IF reversePolarity THEN
    distanceToMoveInSteps := distanceToMoveInSteps * -1;
END_IF

pointToPointAccelSetpoint := acceleration;
pointToPointDecelSetpoint := deceleration;
velocitySetpoint := velocity;

currentLimit := defaultCurrentSetpoint;
_moveDistance := TRUE;

//commands.feedToLength := TRUE;
//SUPER^.ExecuteStoredProgram(1);
END_METHOD

METHOD StopViaProgram
// Load program segment 12 into buffer and execute.  This program contains nothing but a SM command.
// We must do it this way because the normal "stop command" opcode we have access to over modbus 
// also kills the program buffer which is bad.
SUPER^.Stop();
END_METHOD

PROPERTY CommandAcknowledged : BOOL
GET
CommandAcknowledged := _moveDone;
END_GET
END_PROPERTY

METHOD SetTorque
VAR_INPUT
	torque : DINT;
END_VAR
sclCommand := 16#4743; // GC (Current Command)
parameter1 := torque;
															
commandSuccessful := FALSE;
commands.SendHostCommand := TRUE;
END_METHOD

METHOD Execute
VAR_INPUT
END_VAR
SUPER^.Execute();
waitForMove();
_moveDistanceONS(CLK := _moveDistance);
_moveFinalONS(CLK := _moveFinal);

CASE moveDistanceState OF
	AMP_EIP_MOVE_INITIAL_STATES.Idle :						
															IF _moveDistance THEN
																moveDistanceState := AMP_EIP_MOVE_INITIAL_STATES.SetOutputOff;
															END_IF
															
	AMP_EIP_MOVE_INITIAL_STATES.SetOutputOff :					sclCommand := 16#534F; //Output off
															parameter1 := 16#48B2;
															commands.SendHostCommand := TRUE;
															IF commandSuccessful THEN
																commandSuccessful := FALSE;
																moveDistanceState := AMP_EIP_MOVE_INITIAL_STATES.WaitAfterSettingOutputOff;
															END_IF
															
	AMP_EIP_MOVE_INITIAL_STATES.WaitAfterSettingOutputOff :		
															IF commandSuccessful THEN
																moveDistanceState := AMP_EIP_MOVE_INITIAL_STATES.MoveMotor;
															END_IF
																
	AMP_EIP_MOVE_INITIAL_STATES.MoveMotor: 					commandSuccessful := FALSE;
															sclCommand := 16#0;
															parameter1 := 16#0;
															commands.FeedToLength := TRUE;
															_moveDistance := FALSE;
															moveDistanceState := AMP_EIP_MOVE_INITIAL_STATES.WaitAfterMovingMotor;
															
															
	AMP_EIP_MOVE_INITIAL_STATES.WaitAfterMovingMotor: 		IF commandSuccessful THEN
																_moveDone := TRUE;
																moveDistanceState := AMP_EIP_MOVE_INITIAL_STATES.Idle;
															END_IF														
END_CASE

CASE moveDistanceFinalState OF
	AMP_EIP_MOVE_INITIAL_STATES.Idle :						IF _moveFinal THEN
																moveDistanceFinalState := AMP_EIP_MOVE_INITIAL_STATES.SetOutputOff;
															END_IF
															
	AMP_EIP_MOVE_INITIAL_STATES.SetOutputOff :					sclCommand := 16#534F; //Output off
															parameter1 := 16#48B2;
															commands.SendHostCommand := TRUE;
															IF commandSuccessful THEN
																commandSuccessful := FALSE;
																moveDistanceFinalState := AMP_EIP_MOVE_INITIAL_STATES.WaitAfterSettingOutputOff;
															END_IF
															
	AMP_EIP_MOVE_INITIAL_STATES.WaitAfterSettingOutputOff :		
															IF commandSuccessful THEN
																moveDistanceFinalState := AMP_EIP_MOVE_INITIAL_STATES.MoveMotor;
															END_IF
															
	AMP_EIP_MOVE_INITIAL_STATES.MoveMotor: 					sclCommand := 16#0;
															parameter1 := 16#0;
															commandSuccessful := FALSE;	
															commands.FeedToLength := TRUE;
															moveDistanceFinalState := AMP_EIP_MOVE_INITIAL_STATES.WaitAfterMovingMotor;
															
															
	AMP_EIP_MOVE_INITIAL_STATES.WaitAfterMovingMotor: 		IF commandSuccessful AND InPosition THEN	
																moveDistanceFinalState := AMP_EIP_MOVE_INITIAL_STATES.SetOutputOn;
															END_IF
														
	AMP_EIP_MOVE_INITIAL_STATES.SetOutputOn :					sclCommand := 16#534F; // Output on
															parameter1 := 16#4CB2;
															
															commandSuccessful := FALSE;
															commands.SendHostCommand := TRUE;
															_moveFinal := FALSE;
															moveDistanceFinalState := AMP_EIP_MOVE_INITIAL_STATES.WaitAfterSettingOutputOn;
															
															
	AMP_EIP_MOVE_INITIAL_STATES.WaitAfterSettingOutputOn :		
															IF commandSuccessful THEN
																_moveDone := TRUE;
																moveDistanceFinalState := AMP_EIP_MOVE_INITIAL_STATES.Idle;
															END_IF
																

END_CASE
(*
IF _moveFinal THEN	
	IF NOT movedFinal AND commandSuccessful THEN
		commandSuccessful := FALSE;
		commands.FeedToLength := TRUE;
		waitForMove.IN := TRUE;
		movedFinal := TRUE;
	END_IF
	
	IF commandSuccessful AND waitForMove.Q AND InPosition THEN
		sclCommand := 16#534F;
		parameter1 := 16#4CB2;
		commands.SendHostCommand := TRUE;
		_moveFinal := FALSE;
		waitForMove.IN := FALSE;
		movedFinal := FALSE;
	END_IF
END_IF
*)
IF manualFinalMovePB THEN
    MoveDistanceFinal(distance := distanceSetpointInches, acceleration := pointToPointAccelSetpoint, deceleration := pointToPointDecelSetpoint, velocity := velocitySetpoint);
    manualFinalMovePB := FALSE;
END_IF
END_METHOD

METHOD SetRearMotorTorqueValue
VAR_INPUT
	torque : DINT;
END_VAR
sclCommand := 16#4743; // GC (Current Command)
parameter1 := torque;
															
commandSuccessful := FALSE;
commands.SendHostCommand := TRUE;
END_METHOD

METHOD MoveDistanceFinal
VAR_INPUT
    distance : REAL;        //Distance to move in inches
    acceleration : INT;        //Acceleration in RPM/sec
    deceleration : INT;        //Deceleration in RPM/sec
    velocity : INT;            //Velocity in .25RPM
END_VAR
commandSuccessful := FALSE;
_moveDone := FALSE;
moveDistanceFinalState := AMP_EIP_MOVE_INITIAL_STATES.Idle;
distanceToMoveInSteps := REAL_TO_DINT((distance) * stepsPerInchSetpoint);
IF reversePolarity THEN
    distanceToMoveInSteps := distanceToMoveInSteps * -1;
END_IF

pointToPointAccelSetpoint := acceleration;
pointToPointDecelSetpoint := deceleration;
velocitySetpoint := velocity;

currentLimit := defaultCurrentSetpoint;
_moveFinal := TRUE;
//SUPER^.ExecuteStoredProgram(2);
END_METHOD

END_FUNCTION_BLOCK

// FBs/Motors/Applied Motion/FB_AppliedMotionStepServoEIPBase
FUNCTION_BLOCK FB_AppliedMotionStepServoEIPBase IMPLEMENTS IPositionableMotor
VAR_INPUT
    ptrEIPInputs : POINTER TO ARRAY[0..13] OF  DINT;
    ptrEIPOutputs : POINTER TO ARRAY[0..15] OF DINT;
	commFail : BOOL;
    stepsPerInchSetpoint : INT;             //Steps per inch setpoint
    reversePolarity : BOOL;                 //0 = Normal, 1 = reversed polarity for display
    jogAccelSetpoint : INT;        //Point-to-Point Acceleration (AC) Setpoint
    jogDecelSetpoint : INT;        //Point-to-Point Deceleration (DE) Setpoint
    jogVelocitySetpoint : INT;                //Velocity (VE) Setpoint
    pointToPointAccelSetpoint : INT;        //Point-to-Point Acceleration (AC) Setpoint
    pointToPointDecelSetpoint : INT;        //Point-to-Point Deceleration (DE) Setpoint
    velocitySetpoint : INT;                //Velocity (VE) Setpoint
	defaultCurrentSetpoint : DINT;
	sclCommand : DINT;						// SCL Command from 
	parameter1 : DINT;						// Data/SCL parameter 1
	parameter2 : DINT;						// Data/SCL parameter 2
    distanceSetpointInches : REAL;        //Distance setpoint in inches Setpoint
    moveDistanceManualPB : BOOL;            //Move distance pushbutton
    movePositionManualPB : BOOL;            //Move position pushbutton
	isHomable : BOOL;
END_VAR
VAR_IN_OUT
    //slave : IoDrvModbusTCP.ModbusTCPSlave;                    //Slave ModbusTCP Object
END_VAR
VAR
    absolutePositionSteps : DINT; //Immediate Absolute Position in steps
    distanceToMoveInSteps : DINT;        //Distance Setpoint to Drive
    stepServoStatusRaw : INT; //Raw step servo status over modbus
	stepServoAlarmCodeRaw : INT; // Ras Step Servo alarm code word
	currentLimit : DINT;
    commands : FB_StepServoCommands();
    commandSuccessful : BOOL;    //Modbus Command was successful
    commandSuccessfulONS : R_TRIG;    //Modbus Command was successful
    commandSentONS : R_TRIG;    //Modbus Command was successful
    homeRequiredIndication : BOOL; //Home required indication.
    driveInputs : ARRAY[0..13] OF DINT;        // Inputs from drive over EIP
    driveOutputs : ARRAY[0..15] OF DINT;    // Outputs to drive over EIP
    interfaceToPass : IFault;
    faultListRegisterSuccess : BOOL;        // Registering in fault list successful
    _faulted : BOOL;                    // Motor Faulted
	_reset : BOOL;			//Reset Motor
	_homeNow : BOOL;
	homingOSF : F_TRIG;
	resetState : INT;
	IECReferenceGood : BOOL;
	resetTimeout : Standard.TON;
	encoderResetTimeout : Standard.TON;
END_VAR
VAR_OUTPUT
    absolutePositonInches : REAL; //Immediate Absolute Positon in inches
    velocity : INT;    //Velocity (VE) Input from Drive
    status : StepServoStatusFB; //Status of servo
	alarms : FB_StepServoAlarms; // Alarms from Drive
    QSegmentRunning : INT; //Current Q program running from Drive
	faults : StepServoFaultsType;
END_VAR

//{warning 'add method implementation '}
METHOD Stop
commandSuccessful := FALSE;
commands.StopNormal := TRUE;
END_METHOD

{attribute 'monitoring' := 'variable'}
PROPERTY Homing : BOOL
GET
Homing := status.homing;
END_GET
END_PROPERTY

METHOD HomeNow
commandSuccessful := FALSE;
parameter1 := 1;
pointToPointAccelSetpoint := 50;
pointToPointDecelSetpoint := 50;
velocitySetpoint := 500;
distanceToMoveInSteps := 0;
commands.sendQAndExecute := TRUE;

//homeRequiredIndication := FALSE;
END_METHOD

METHOD MoveDistance
VAR_INPUT
    (*Distance to move in inches*)
    distance    : REAL;
    (*Acceleration in RPM/sec*)
    acceleration    : INT;
    (*Deceleration in RPM/sec*)
    deceleration    : INT;
    (*Velocity in .25RPM*)
    velocity    : INT;
END_VAR
//This method preps the data to send to the drive and triggers the send.
//Set distance and unpack to prep data to send to motor

commandSuccessful := FALSE;

distanceToMoveInSteps := REAL_TO_DINT((distance) * stepsPerInchSetpoint);
IF reversePolarity THEN
    distanceToMoveInSteps := distanceToMoveInSteps * -1;
END_IF

pointToPointAccelSetpoint := acceleration;
pointToPointDecelSetpoint := deceleration;
velocitySetpoint := velocity;
currentLimit := defaultCurrentSetpoint;

commands.feedToLength := TRUE;
END_METHOD

{attribute 'monitoring' := 'variable'}
PROPERTY CommandAcknowledged : BOOL
GET
CommandAcknowledged := commandSuccessful;
END_GET
END_PROPERTY

PROPERTY InstanceName : STRING
GET
END_GET
SET
END_SET
END_PROPERTY

(* This will be called if the machine is faulted*)
METHOD MachineFaulted
END_METHOD

METHOD MoveToPositionTorque
VAR_INPUT
	(*Position to move to in inches*)
    position    : REAL;
    (*Acceleration in RPM/sec*)
    acceleration    : INT;
    (*Deceleration in RPM/sec*)
    deceleration    : INT;
    (*Velocity in .25RPM*)
    velocity    : INT;
	(*Current in .01A*)
	current : DINT;
END_VAR
commandSuccessful := FALSE;

distanceToMoveInSteps := REAL_TO_DINT((position) * stepsPerInchSetpoint);
IF reversePolarity THEN
    distanceToMoveInSteps := distanceToMoveInSteps * -1;    
END_IF

pointToPointAccelSetpoint := acceleration;
pointToPointDecelSetpoint := deceleration;
velocitySetpoint := velocity;
currentLimit := current;

commands.feedToPosition := TRUE;
END_METHOD

{attribute 'monitoring' := 'variable'}
PROPERTY InPosition : BOOL
GET
InPosition := status.inPosition;
END_GET
END_PROPERTY

//{warning 'add method implementation '}
METHOD Disable
commandSuccessful := FALSE;
commands.Disable := TRUE;
END_METHOD

//{warning 'add method implementation '}
METHOD Enable
commandSuccessful := FALSE;
commands.Enable := TRUE;
END_METHOD

METHOD ResetEncoderPosition
VAR_INPUT
	position : DINT;
END_VAR
sclCommand := 16#5350; // SP (Set Position)
parameter1 := position;
															
commandSuccessful := FALSE;
commands.SendHostCommand := TRUE;
END_METHOD

METHOD Execute
VAR_INPUT
END_VAR
//    Function Block: AppliedMotionStepServo
//    Description: This block provides an abstraction for a Ethernet I/P Applied Motion Step Servo
//    Created by: Ben Hess
//    Created Date: May 11th, 2018

// Use pointers for EIP memory register locations
driveInputs := ptrEIPInputs^;
// Step servo command bits handler
commands();
ptrEIPOutputs^ := driveOutputs;
alarms(alarmCode := stepServoAlarmCodeRaw, faults := faults);

IF currentLimit = 0 THEN 
	currentLimit := defaultCurrentSetpoint;
END_IF
//Map raw EIP Registers to parameters
absolutePositionSteps := driveInputs[5];
velocity := DINT_TO_INT(driveInputs[8]);
stepServoStatusRaw := DINT_TO_INT(driveInputs[0]);
stepServoAlarmCodeRaw := DINT_TO_INT(driveInputs[1]);
driveOutputs[4] := velocitySetpoint;
driveOutputs[5] := pointToPointAccelSetpoint;
driveOutputs[6] := pointToPointDecelSetpoint;
driveOutputs[7] := distanceToMoveInSteps;
driveOutputs[8] := currentLimit;
driveOutputs[9] := sclCommand;
driveOutputs[10] := parameter1;
driveOutputs[11] := parameter2;
driveOutputs[12] := currentLimit;
driveOutputs[13] := currentLimit;
driveOutputs[0] := commands.commandWord;

//Convert Distance setpoint to steps.  Reverse polarity for display purposes if needed. 

absolutePositonInches := (DINT_TO_REAL(absolutePositionSteps) / INT_TO_REAL(stepsPerInchSetpoint));

//Homing required from motor - for now just if there was an initialization seen.
homeRequiredIndication S= status.initializing OR Globals.firstScan OR _faulted OR driveInputs[11].0;
//homeRequiredIndication S= status.initializing OR Globals.firstScan OR driveInputs[11].0;
homingOSF(CLK := status.homing);
IF NOT driveInputs[11].0 THEN
	homeRequiredIndication := FALSE;
END_IF

commandSentONS(CLK := commands.commandSent);

IF commandSentONS.Q THEN
	commandSuccessful := TRUE;
END_IF

commandSuccessfulONS(CLK := commandSuccessful);
IF commandSuccessfulONS.Q THEN
	//parameter1 := 0;
	//velocitySetpoint := 0;
	//pointToPointAccelSetpoint := 0;
	//pointToPointDecelSetpoint := 0;
	//distanceToMoveInSteps := 0;
END_IF



resetTimeout(IN := _reset, PT := T#1S);
encoderResetTimeout(PT := T#150MS);
IF resetTimeout.Q THEN
	resetState := 0;
	encoderResetTimeout.IN := FALSE;
	_reset := FALSE;
END_IF
CASE resetState OF
	
	0 :		// Do Nothing
			IF _reset THEN
				resetState := 1;
			END_IF
	1 :		// 
			commandSuccessful := FALSE;
			commands.alarmReset := TRUE;
			resetState := 2;
	
	2 :		IF commandSuccessful THEN
				commandSuccessful := FALSE;
				commands.Enable := TRUE;
				resetState := 3;		
			END_IF
	
	3 :		//
			IF commandSuccessful THEN;
				
				encoderResetTimeout.IN := TRUE;
				IF encoderResetTimeout.Q THEN
					resetState := 4;	
					ResetEncoderPosition(driveInputs[5]);	
				END_IF
			END_IF
	
	4 :		//
			IF commandSuccessful THEN;
				resetState := 0;
				
				_reset := FALSE;
			END_IF
	
END_CASE

IF reversePolarity THEN
    absolutePositonInches := absolutePositonInches * -1; 
END_IF

//Get Servo Status and unpack
status(statusCode := StepServoStatusRaw);

//Bit-packing for LONG types over Modbus
//_faulted := status.driveFaulted OR status.alarmPresent OR commFail;
_faulted := status.driveFaulted OR commFail;

//Manual moves for motor
IF moveDistanceManualPB THEN
    MoveDistance(distance := distanceSetpointInches, acceleration := pointToPointAccelSetpoint, deceleration := pointToPointDecelSetpoint, velocity := velocitySetpoint);
    moveDistanceManualPB := FALSE;
END_IF

IF movePositionManualPB THEN
    MoveToPosition(position := distanceSetpointInches, acceleration := pointToPointAccelSetpoint, deceleration := pointToPointDecelSetpoint, velocity := velocitySetpoint);
    movePositionManualPB := FALSE;
END_IF


faults.commFail.faultTrigger := commFail; //AND Globals.machinePowerOK;
//faults.notHomed.faultTrigger := homeRequiredIndication AND isHomable;
END_METHOD

{attribute 'monitoring' := 'variable'}
PROPERTY HomeRequired : BOOL
SET
homeRequiredIndication := HomeRequired;
END_SET
GET
HomeRequired := homeRequiredIndication;
END_GET
END_PROPERTY

{attribute 'monitoring' := 'variable'}
PROPERTY ActiveStoredProgramNumber : INT
GET
ActiveStoredProgramNumber := QSegmentRunning;
END_GET
END_PROPERTY

METHOD Reset : BOOL
VAR_INPUT
END_VAR
_reset := TRUE;
END_METHOD

{attribute 'monitoring' := 'variable'}
PROPERTY Faulted : BOOL
GET
Faulted := _faulted;
END_GET
SET
END_SET
END_PROPERTY

METHOD MoveToPosition
VAR_INPUT
    (*Position to move to in inches*)
    position    : REAL;
    (*Acceleration in RPM/sec*)
    acceleration    : INT;
    (*Deceleration in RPM/sec*)
    deceleration    : INT;
    (*Velocity in .25RPM*)
    velocity    : INT;
END_VAR
commandSuccessful := FALSE;

distanceToMoveInSteps := REAL_TO_DINT((position) * stepsPerInchSetpoint);
IF reversePolarity THEN
    distanceToMoveInSteps := distanceToMoveInSteps * -1;    
END_IF

pointToPointAccelSetpoint := acceleration;
pointToPointDecelSetpoint := deceleration;
velocitySetpoint := velocity;
currentLimit := defaultCurrentSetpoint;

commands.feedToPosition := TRUE;
END_METHOD

METHOD SetTorque
VAR_INPUT
	torque : DINT;
END_VAR
sclCommand := 16#4743; // GC (Current Command)
parameter1 := torque;
															
commandSuccessful := FALSE;
commands.SendHostCommand := TRUE;
END_METHOD

METHOD ExecuteStoredProgram
VAR_INPUT
    (*Program number to execute*)
    programNumber    : INT;
END_VAR
parameter1 := programNumber;
commands.SendQAndExecute := TRUE;
END_METHOD

{attribute 'monitoring' := 'variable'}
PROPERTY CurrentPosition : REAL  //Current motor position in Inches
GET
CurrentPosition := absolutePositonInches;
END_GET
END_PROPERTY

{attribute 'monitoring' := 'variable'}
PROPERTY Moving : BOOL
GET
Moving := status.moving;
END_GET
END_PROPERTY

METHOD MoveDistanceTorque
VAR_INPUT
	(*Distance to move in inches*)
    distance    : REAL;
    (*Acceleration in RPM/sec*)
    acceleration    : INT;
    (*Deceleration in RPM/sec*)
    deceleration    : INT;
    (*Velocity in .25RPM*)
    velocity    : INT;
	(*Current in .01A*)
	current : DINT;
END_VAR
//This method preps the data to send to the drive and triggers the send.
//Set distance and unpack to prep data to send to motor

commandSuccessful := FALSE;

distanceToMoveInSteps := REAL_TO_DINT((distance) * stepsPerInchSetpoint);
IF reversePolarity THEN
    distanceToMoveInSteps := distanceToMoveInSteps * -1;
END_IF

pointToPointAccelSetpoint := acceleration;
pointToPointDecelSetpoint := deceleration;
velocitySetpoint := velocity;
currentLimit := current;

commands.feedToLength := TRUE;
END_METHOD

END_FUNCTION_BLOCK

// FBs/Components/PrinterFB
FUNCTION_BLOCK PrinterFB EXTENDS BaseComponentFB IMPLEMENTS IComponentStatus
VAR_INPUT
    autoSendLabel :BOOL;    // Automatically send a label                
END_VAR
VAR_OUTPUT
    state : PRINTER_STATES;         // Printer State Machine
	oLowerPrintHead : BOOL;
	printHeadDebounced : BOOL;
	
END_VAR
VAR
    _amPrintNow : BOOL;                // Auto mode - print now
    _amSendPrintSignal : BOOL;        // Auto mode - send print signal
    _amGoToIdle : BOOL;                // Auto mode - Acked, go back to idle mode
    printHeadDebounce : TON;
    printHeadDebouneSetpoint : TIME := T#50MS;
    tcpServer : FB_TCPClient();
END_VAR

VAR_IN_OUT
END_VAR

//    Function Block: Printer
//    Description: This program manages the aspects of a (Zebra) printer
//    Created by: Ben Hess
//    Created Date: April 2nd, 2018
SUPER^();
// Enable TCP Server for label sending
tcpServer();

//Report as ready if mode is auto and we're not faulted
_ready := (_mode = DEVICE_MODES.Auto) AND NOT (state = PRINTER_STATES.Fault);

printHeadDebounce(PT:= printHeadDebouneSetpoint, Q=> printHeadDebounced);
IF enableONS.Q OR resetONS.Q THEN
    state := PRINTER_STATES.Idle;
	_reset := FALSE;
	_amGoToIdle := FALSE;
	_amSendPrintSignal := FALSE;
	_amPrintNow := FALSE;
END_IF

IF NOT enable THEN
    state := PRINTER_STATES.Fault;
	oRunPrinterRibbonUnwindMotor := FALSE;
	oLowerPrintHead := FALSE;
END_IF



//State machine for the printer
CASE state OF
    PRINTER_STATES.Idle :                            //Go to waiting for data if printer is ready
                                                    oRunPrinterRibbonUnwindMotor := FALSE;
													oPrinterStartPrint := FALSE;
													oLowerPrintHead := FALSE;
													printHeadDebounce.IN := FALSE;
													IF NOT printerDataReady THEN
                                                        IF autoSendLabel THEN
                                                            tcpServer.SendLabel();
                                                        END_IF
                                                        state := PRINTER_STATES.WaitingForData;
                                                    ELSE
                                                        state := PRINTER_STATES.DataReady;
                                                    END_IF
                                                    
                                        
    
    PRINTER_STATES.WaitingForData :                    //If printerDataReady drops out the label data was received
                                                    
                                                    IF printerDataReady THEN
                                                        state := PRINTER_STATES.DataReady;    
                                                    END_IF
                                                
    PRINTER_STATES.DataReady :                        // Wait for command to begin printing
                                                    IF NOT printerDataReady THEN
														state := PRINTER_STATES.Idle;
													END_IF
													IF _mode = DEVICE_MODES.Auto AND _amPrintNow THEN
                                                        state := PRINTER_STATES.BeginPrintCycle;
                                                        _amPrintNow := FALSE;
                                                        oLowerPrintHead := TRUE;
                                                        oRunPrinterRibbonUnwindMotor := TRUE;
														//oPrinterStartPrint := TRUE;
                                                    END_IF                                    
            
    
    PRINTER_STATES.BeginPrintCycle :                // Start printing
                                                    
                                                    printHeadDebounce.IN := TRUE;
                                                    IF printHeadDebounce.Q AND _amSendPrintSignal THEN
                                                        oPrinterStartPrint := TRUE;
                                                        state := PRINTER_STATES.Printing;
                                                        printHeadDebounce.IN := FALSE;
                                                        _amSendPrintSignal := FALSE;
                                                    END_IF                                                    
                                        
    
    PRINTER_STATES.FeedAtPrintSpeed :                //

                                                    
                                                                                                
                                        
    PRINTER_STATES.Printing :                        //While printing, wait for End of Print signal
                                                    IF printerEndOfPrint THEN
                                                        oPrinterStartPrint := FALSE;
                                                        oLowerPrintHead := FALSE;
                                                        
                                                        state := PRINTER_STATES.DonePrinting;    
                                                    END_IF
                                        
    PRINTER_STATES.DonePrinting :                    //Done printing, feed a little more through
                                                    IF _mode = DEVICE_MODES.Auto AND _amGoToIdle THEN
                                                        oRunPrinterRibbonUnwindMotor := FALSE;
                                                        state := PRINTER_STATES.Idle;
                                                        _amGoToIdle := FALSE;
														HMIData.printerCycles.Increment();
														HMIData.printHeadClean.Increment();
                                                        Globals.printerCycleCounts := Globals.printerCycleCounts + 1;
                                                    END_IF
        
    PRINTER_STATES.FeedThrough :                        
                                        
    PRINTER_STATES.Ready :                        
                                        
    PRINTER_STATES.Fault :                        
                                        
END_CASE

METHOD AutoSendPrintSignal
VAR_INPUT
END_VAR
_amSendPrintSignal := TRUE;
END_METHOD

METHOD AutoPrintNow
VAR_INPUT
END_VAR
_amPrintNow := TRUE;
END_METHOD

PROPERTY Mode : DEVICE_MODES
GET
Mode := _mode;
END_GET
SET
_mode := Mode;
END_SET
END_PROPERTY

METHOD AutoAckPrintDone
VAR_INPUT
END_VAR
_amGoToIdle := TRUE;
END_METHOD

PROPERTY Ready : BOOL
GET
Ready := _ready;
END_GET
SET
_ready := Ready;
END_SET
END_PROPERTY

END_FUNCTION_BLOCK

// FBs/FB_TCPClient
FUNCTION_BLOCK FB_TCPClient
VAR_INPUT
END_VAR
VAR_OUTPUT
END_VAR

VAR
    // =======================================
    // set up Client
    // =======================================
    _TCPClient : NBS.TCP_Client;
    _TCPClient_ipAddr: NBS.IP_ADDR;
    _TCPClient_uiPort: UINT := 9100;
    _TCPClient_hClient : CAA.HANDLE; // Client handle
    _sClientIP : STRING(15):='192.168.10.160'; (* this device's Client IP address *)
    _uiPort : UINT:= 9100;
    _TCPConnection : NBS.TCP_Connection; // TCP connection instances
    _TCPConnection_hConnection: CAA.HANDLE;    // handle of client connections    
    _TCPWrite : NBS.TCP_Write; // TCP write
    _TCPRead : NBS.TCP_Read; // TCP read
    _sTCPSendData: STRING(25000); // This is the label
    _sTCPReadData: STRING(1000); //receive up to 1000 chars if needed
    _TCPWriteEn: BOOL;
    _sServerIP: STRING(80);
    _sendLabel : BOOL;
	label203 : STRING(25000) := '^XA~TA000~JSN^LT0^MNW^MTT^PON^PMN^LH0,0^JMA^PR8,8~SD15^JUS^LRN^CI0^XZ
^XA
^MMT
^PW812
^LL1218
^LS0
^FO0,0^GFA,129792,129792,00104,:Z64:
eJzs3T9v5MYVAPDhcr2jQlkqRoo1LIvKOR9A6VQox72LArhMFxcBIsP5AHJ3xUGc3TVOFyCxXaRwlSKfI4ApC7BTJHGbLhRcqAwNNzTCcPLe/OOQnNXpdBR15/AZ0Z9dcn5L8r3hDEldCBliiCGGGGKIIYYY4uWNWU/O47t3As7Lzhx+FcN53hHjcbb2HRGp+DAQYjmf622k1aeI5ZLqN1/9Vt8VlCd37ITVymJVsZzYl8T8lFsfSDftm19Tq7XgMlvj6KWZWpXp1su1jmi5cnCVQG1WuFpzpAO9cOZ2QpdT1p0cF5PNxaS4Wye0FnY5Mb5WNBxslFa/wduZl4rFS5CcYS9Ma0flKietOZyAIhwvJxFzMdbKthPqxgk3jrWjcCfbTuJ9VezhMjQjQXKXTi07HY7ndvK6k/rT6bbY3ylSjgiqhROXQ91OWVuTZ/7UF07IiO8soNDeF2sd3nR43SlG05FwYnLpTuy+nMh2At26eDmz9qtFymB1ZxrsTHGZ0rtkzgKynNzlhNdyymlQoOPl9DJxFpC18HM5qf0JwZnuoUMz6K+dif2yOLHeTVc63J9uYx4EaXiZuwpIlqFsohCr5oZPrc9xTSdk8WXhKiDhZPJjP8sJ7YazpjM9wK0n/JK7ErtXhxF1ZNqO7ma1U6pjB04sF5ZLnP1jiv1o6YHjKiCxlNr3Loc2nKLaB7HcE3KRRJx/oHzAcRWQrxxPtBHrveU1ncRySN2Rg6QDPxFpDY4rsft0yjUOLh1YTsStmqocuawYh0D5gOMqoMopVQN1J7zaScyyPm4plA84rgLS+02G2/nY7fCaI9eHFy+5K7HvzklqTvxcDpQPOo4C8nViiTBrGB6/B6p9s7XrHCwfdBwF5HP9ITtwMK3RcSR2r445QC1HlJXbMWPxysHyQcdRQNLJmo6eZmF3kLccXnOqyRmWDzqOAlL9MbNQHeWVTlp3xPqY1ug4ErtnJ1/jCCLg1Ykm0etUDjUOlg8/5a4C0uex1O2ELsevHFwr0j+I8uH4uqOAdKvrnaTphGJL9GZ4elmZ1iXhzsTuy4lUq+YMXHNibJrWHbmrGW0uK8snx3UcBaQd3nIKtbVMjh0aW0vajiifbCtyFlCoF03XOeQajsjjCBdPZ7ib24ltRv25w/HWOmVtuiAdkdbsMS7OTu7KqebbDkfO71xOXnfEeESUD3lWATVmTmbqbpzap2g4KVaFSGuPM+5M7FAvm7QdWTlq1krrb9YWTkxaU57E+C29K8dfsyo64Vonrc8e0AkFEPAschaQOUC528mcTmOWgu2I8slCeR7x2kMr3XpRn9HgsY3FN7/tlHWnSus05oU7sXtziFm45XDbsRvO6r/iwfBk+3ztGchkQstRkz115rQbZtVFZgxMA1E+3FNWFibtDYqf1ylJ3WE6rUvcpjWJ3Z+jBz32quioU2bbyeqOqJUwifTYKHIXkE454aQGTvRoUTnW1qZ1RxxyXT4SKx0FpFPO7Zi2LKe+PfKI67Tm6xO7Pyd0OqHlJE2nEuQxLnD3MvH2ugJStS6cxHLilmP61pZTlY/UUlcBqQw2q6qxZt1RW7vGqdL6isTuwYmqoXnL4S5H33loOFX5uAoo1Au7HO8qR1/oMp/XlI+rgEJu35i7ykm147udKq1did23I9ZamVXlmdpf6/CWY5ePo4DQydY59RGani64Hbt8HAWkHXp9RwH6QqQKO60did2nU2jHbzih7eQNh9Ydu3wcBRTyan7Iqwm6HFFH65206djl4yigUK2M34pq1dDh1C75tBw7rR2J3aujBgYtx2acTrVj6uXTLqDaPamGU+sOLAc30771hVEvn3YB2U5+pVNc6dTTup3YfTm1W7yNu0zVpdNY79VSv5k3nHr5tAvIdpKGI9ZibSd0OPXyaReQd2NHftVRT+t2Yvfl2DXCGo7YC+bXypEn7pojyyexGmsWUGTeKa27TPhTGumGxa+lKUyH0ywfzhe8XkCheSe3nNjhhLbD6w5tpHU7sftyrJRvOry2GytHFmzMrev4onyK2gMJ+IJfXe2zuqSGc/EcTrN8YMWwcQbSb5TEWtU42TqH1ZwTT+9otfvXJ/ZtO3pjM8sRO/Mcv6TG4Z/p3ei1HKt89Ay5lAVUOfoAkabz1ZVOyi3Hz035mMFTs4DUBqXkBUKmdTWMwR/kxSur2b4cK51vGlX54PkiM92WXUBdRCSv6OAXPEjyMmS49iLCjaNKayaee/JNYnf3uGiPjlU+BCvzMXEV0IuHL0ZKnqhSPPCBqMRWAb1wVGmdU4b9khgBYGKntcR+VRy5c+QtQ4JVmlFd+bqAYv7iwahsEtuegaee2xQvqu3xn9XGdSLxTffKjuVz0WLyUG1qb07YhZN6BbaDRUOgSsWewhSPsXa7OzzQd56Iq7wR9GeMhKphWbuyP/Ce1cS1AiaYeEUAkrukhDwSLUdylrMoenU6SQMcA59xMe7Pp0Q9TRxxWbuyfOizmrheQAFxMeHLdggVaQZFK099qXZSD4cULKR5mMPGEk4XfCVuxmf+GV9ksN4mrBznFOeRzE9h8YLEzOPYv9A8SikmdiTuAGYzMiXKwQFRrtK6LyfE3iFKo5IENAthcJSQGNpccWiGJ17KKfOkE+GYPIbXs+gMnIARdOCMEDG/KqD0WKUBoXLipconEvfzkihHJ4YDyaRTYiYSdIh2MooXSBmRDmxlTPwCnPvAQQGJDjoCR/WbVJbPSeUU4GThv+FQguMXHJ2Cfgszsv+mMaXfcQoDGXTOypiv0j3IrSKkiyymMGz6Nr9P/4OJLTrOiKUq3eAzWGntcmLpfNOpA4cqLYMkzGLYDDhrwJufwT5a5WHJSxiInUxhf2gHa3GVHYQ+OItFHlKY45T5QVgVEGepSmtwrPJRzjSEjIM0Oz/FoZ5wMH1qTuB0Yi4cVUApXzBKVOD0oqBp26HgYPt0Ga1wgg5OMdtRzir4XDn3gdYOjHCkk/g4fUu5x6a2o9O6dwemVJPKCaXjo0MrZ+F2xFBAFBA6M+NQkRimG03L6TSAJibQ2CqPpSOmcvhkZOxVDo5fVhlOtIUD+QYzsfy+GOYQ2HqYAHrk2HZ0+SgnRAdWPz3P0FmdrjB7OInwTzhi6dAvaAIfeZVqB/N6hQ7uFJnYZ3BaMA6e+nRa9+oUO2scGOwRvOZDoZtZnT6h2LdCvwf9PdSp6N/QiZgpIHRSyyn19Tc5ytoJfeUkWcwiuvpydYYPL0G70DNS4+AFbCbOK9i/UXQKkkfiaSWYJgjHY5Zjykc6B9qhyjmXToZPlMAX7RSiv8bpB/bXnnbEc2MisWtOfFqlda8OpL4v87rhwBlkgV9EHpx/RPHMtcLTHJ7nFnDO4MIpdCvgTEy3g44uH+nwIjpfiDoNsizOwbmAPMD+KsEpDFPOlOKWrLIInZBLhydQ2QtdQE1Hl49yMuJdYL8DQ7pHyrngql/EL8bJbScTdYoOJqdIbHCmtqPTujfH0444L6ATSSeNr+UkxhEF1HDK6vJ1bDnMOLnfdrL7VzocJjp154Sa8lEO/Ifn0zSP8oNAOnn0TEee54yDiQ3OzHLyag7cu4PjENhpBz46BczTobUI6yf2jPOvxNSPdoIkv38ib0NAAUGd2k5aXb2OlCPGbzM4OPASOpAoHMdwC/wi+oPsBIdsMH6rHPH3XvmBfrK6DBpOUl1MFM4FbD84+SwugkQ62B7eDl7gM3bCycHxRH+tnDLE8Sg6YjKAiZ2U9NhyFtbdFHTOwMHxNQGngPH1Cs7YePMKzjcLGHgbB7pu7K+1E4CTwfiaRVwldt2ZWHdlenS6CiggGIdYzrgqn67mWRiQ2Lvcqy4fFjPrElI380YRkNik5th/HtqX0818WwQUEImqYQg49uMUcWcOfH7YAuP4ee0SbNSZU+K80HZqj9X05XSY2HhLmB1VjlU+nSZC6mdhahzqfA6yk/Ay62IoOOwVd0gRVGUaJPdviyEHtEqxIDm4NWfbciK2/8o7U6+6OxJXpdR5jIjlkOTWHM/6p0OKaibUefg9OV4S68bdf8rfWYSp+oHermM6hKDb+5l35ZjdFSW36phCNQlxS8Eb3191J07FN9rtbe12hDLPgtstH/OP48TJ98Tx1B+Kslt2iHgwI7jtNMAZIhM3UL4vjhywJ7fuyAd4b58h+m+Wvy8O3tnug4FMYL04QwwxxBBDDDHEEEMMMcQQQwwxxBBDDDHEEEMMMcQQQwwxxEsUx2Tkl4yQA7JB5urBJXxuZX8cULLKLor97U6c35MR2YV2H8LP89FYvDaH/x1u/nBjsfRmG4f3umC8sXIWwhkZZ/mj3U+Wy9HGxvJBJw557Uu2+5dtj3zyzv6D0ejXH2z8is3p1nz5E8KWH47IVkfO8eQe2f38HjqHD0fjo99tvDufbzxlyzFZjE8/T7cOu3Gejl8nu8sH6CwP/eLB+I+fzOOtX5Dl2KPjD9/e2t3vxhlXDntnNBbOXDrkKXt9Y/fw7Q6dWDjvjkYPxn9G5yE4I/JLdJZvdejMhfNb4+D2jMlvUnS8Dp0H5A9wfB7WnI2t+Yevb8y7yTfyFPNteY/8fOuvmG/zpw+2RL4djrdmbPnjrXk3dUqOXztnu8tt8rOPoX78fH6MDtTP/jg6JYskne939GjwuJtm/u+cIV7q2MEvHv+OEfm88Yz4hETmGaZYnMkjMvOzgHkL7mVxvkNu8AQajgVmysHnDKVjHmKSTsxmNA9Tf8H9PM7jxQ3+HZ+LBNueiAe0d/Dfg0Fnb1O/faQWejTd3j+mKzLZJnsX56fP7ySWM/O1M6k7SZLPpsd74GxOyVHypf9izp742nY89v4/Z5OjvR+AMwHnixs8np4kk0cxOH/ycnCeTGbhioLz5ukFY3/LwImm8CHe/5RMyN5bK/y/OU1u5LzHJgU6n/kFNPrFZBadT8EJP/5mkfw9h5fiJ5seO4JNJkdvrB6/kZHkvSc3cCJCP8L99vXpVDrHX8Oh3tze3j87+2obXro43xbOJk1+elq+mXssmtzAiRml6Jw9odJJ398nUT7b3z5/76NNEn+TfP2pctIPTv0dQONT/3mc/wEAAP//7N1BbxvHFQDgmYyy4waLXfuSrKEt99jrGi2SCSyIPhTopUD/wgoG7GM3yIVA1XIEAtRFUK4+9NCf4NxyHIJAfQmsaw4FPKqA5FIkaxgoNgjD7XszS2ol2yKpehetMCODIi1qP+7uvPdmCHHW/psoj6FzcMSso1gO8ROl/nTvCB2599Q4EUn3JPtrwMhkerixQ5WunS+qhaNJGoDz8KHvkwwMbZyURBNJn3iMqtOfN3dk9ppTkJSB8+jXF5yM3DUOnJzsx//COcL4MY6wzsefNB2qyN1K187m/eCicw/iRz2Ma+dj69jzw2R2t/rWOo82zwewCe4Z55iRqD8OoL/56Ij4Nx8aR519BaEZeSQX9JD5PkTT42vkHa1s/BwcepBHeS/Kpx72g1jEMToQPxHk0QjwnI54EPtET73V273chpAPEnRGM8Kr0b+jPuSd/jwKi9qBfIB1IZknmh7MeQmPRtf429c+8QYhOgcloT9Nvo0SxiTEKddwiHyT3wKsc8kc6pwsaeHDo2v9pXXzIKjrbOAaTpvNOa7hqMMsqfaAVTOFd7g2RzKDsaNePIfbu1wRxXWoIJhwkYkZV1xt4JiPn6iFg0PE2lkOSmsngbFBUiSaiKQMi+EM7q//t/ch0bgRBRs3zsAMhNE5/+xl3VOEYEoIkZNBSmJBbkWpWP/jmQlRWdPRfOks3xCrnTTiKo3ziJQpETG5nUZpdHlzb23Diw5VdoyBznLwu3QSlflQWr9JcWScplF2a23nFZUpORmVsLETmcDW6ZiOmc4EOJ+MtHrwaB+d/RiGKf4OODDqfwIOvBRw/NVA3abovDhDp9JDZZ2wyHJw+l+USj+q4Ee0wgGvnyoCDot+hcfgwUYOQ6fI8bgVmdZQKf9Ox7HAQQGWOqUfj6RH2GgMw0ifoJPzaFg8hD4epZs6OkUHbjPrRPEe7JkQkZ/97RlFhx7G1omYDqKB+GNBZag3dZQw/eCeTK0DgzcJ8ZOKYO8pDNp5dUihehtHsMKPMpCoTIp0/fdorRNdcshjOCVlmnp7XxpnTCZPrQNdOoJBcA5zJYil9d+TueBUxcIZYvyAc+/LMR43j0wK62QkhqjxM59hP//Xu3ACdO7UjtLWUbgv1sl8fnTN44bxY5zPYdDhgXN/++L+4MJ9wzk62M/Jpv2g6YyxH2B/Q2d726sde35g8gJOtnDWzzsM845KraMg77xqOCKoHU6nT+B8EGWiCOIzNU62oWPjBzQIpaHHxlGEcRqkkf/BB94yftCJ8DbCDAoJLso3caAuFJl1Ck0GCeOYDzLsb3EcBNYZwagUqgC8ELiNRBoJfCzy1cDSgTr3QpXGGeLFjEY/2/wG8ROWtWPyG9Y5rG5QT4sQxqWm5q3vQN0+kQPjJJLwl+pHm68rnTK9tWUcyNfc1G2s1iTCiu3D41Cu7Zim3vrg3bYWN+2c/yOni6boclnSUps75iqmsfnHmivM88Unc+eQblmJSwdFYaUSZVYkX7GCDFXcfCz+9rmTzBpOYyq6cFglmQzxUpdEgIOruY0qMrx6DMxUaD7SmZ87/XnDaUytFw6vFJdJhfs6AKcq8Wq7asXHkLlKzKgfMqKoF1Tat4syG0c2RgCL5f74CBLObnh4oEkZE1oMCOOjSTG40glVbFZ3bThFvQyrcXqvOyHViRTshBTGUTvEC+mpunrs01d28w1Hs4Zzvibe0gmgSMmcPic5BYcB4AfkbIXz59ccqqha5fwEjiI5QwdeVAxO85lvaJ/BNjV9Npmjc1bQ0jg6iFkRc+hXQTBIDlQenxXocD1gMF/Jz2AkAQ7/yjpitbNnnBenxvmh5HP4RarBCWdxCPfjoByegvNDiU5S7nDYz3xqHM1FPMO9TEO6yoGnU3BeGgevpoAvEJ1kHvewv4VF9VKVMS4LirNKwMGB5zAFI22xXXEodjkfTddwFC0H5vzMdhM8VsbZ7cW4Cl8ZHhSlLsVsF5393V5v4chE9US/Ouxr6DnVqNkz3+zggRLGKXoxWzgijAfGoUrobwQupl3pPAjj2uHQVXfELn8GiUDTiqqVDgdnxzqBMBNHdAY8LjAfBEztoBOgU4R8p3ZC0tcw4qHPdIm5a1K88cqNTSeEm9j264aTk19qjNMA+sLeP3JtHM0hf1oHXn6RC0K/k/A7IdPV96ucXsPpV+dOgk6AzmdfGwdn46yoHUhIgwLm9d/JGKNMD5+vcnbe5sBxk9w4R0sHkpR1IJ19qtEhsQmp5HiVM7jkKLqOA2XgU7xwycIhq/o1/Gbj/JBFPshJb7Bw7h/ry8eNqXPHhC65Or/BeVeXnT3jcIyf2hk3nQAzLYdzAg7kqnUdqAKL+NEBlhv9J6l72K9j66id+17tQL8W1gmhmw5gKE+n0qSiz+UqJyQNJ4bzVfQlBKwITN4JAojTbU9ZB+J0B+sP1iVcVlnEdKoEJ1gXrn5PiWLdoEVZO7iGMtTT8i+Yd0ITP/BDKLnW2d8NelhPmRSEHxRE9PiBLgMSHpzqq+s2VQmujo/RjE5oLtgkh9/HyQyOO+YDUhVLB/Ioxis4/WoK4wMYh8jKpIrJinUwqOqD80LvWoebS0Wr/vM4LLH+4MUIhhr6gnWgLoR2vDOELSsioI7Aj/G/VlzjxzonmG3RwcEcf1kkx1jnIPVXsJFELh2oc3BgsUYNYUAFvwJ1McGKMG8uOHkFdvHx1S/t+u2y01ZzjnNcc80111z7n2/vbvnjuknnOMc5znGOc5zjHOc4xznOcY5znOMc5zjHOc5xjnOc4xznOMc5znGOc5zjHOc4xznOcY5znOMc5zjHOc5xjnOc4xzXXHPNNddcw8Ztfbgxjl1xk694lnOc844cSuCrPWdAiFkOreX9oTNc4qgDZzwj3h3ZusPYMdm61YXjdeZ4v+jGYa9IJ+eH/hMFiq3V/mZaB/HThUMWa/N1lt9uE/i6Qfn65jjmWj4tx8/S6WB/3rvVjbO11b4zrPTCwQD6qE3H80n7+U0qc7Gq1usCrp9fdONYod34MU4H/Y3JjPAuxm8TBY5sP04rVcfPbWytxQ8Z1t9vUF3oxsnst9brT+203a+rbsaJrJp345jjJluPn3PHPGy5X98sx+TRDsZvneRr026i03L9MTsiO9gfr/mtVaeb/uZ1FD+wIx3MS0xd6GKc2JFjgC7Gb9gPOpmfgtPB/KfLOLXCHWwtnh/SyXwOWyfzU4gf7/fdOFu/Je3HD5W1Yx61eH5UJ8cN5wts0I1D8dpTrcdPZr+1vj+6E4fBvL4bR9o7HeQ3027MvL4jB993Me9ft3x+oB9QnHK3/f7B14owvOiz9wDb79py2JG2l6ZvO378DIZvsvXzs3Q62J/3O3J4Bw49UuQ97Actnx96Igk3/do8bC8f/IGQ902cths/2LZWzRf+AwAA///cnUGM28YVQIc7WzFAFDE+GN2gyjJ1DwWaQ2UYCFTUWPng3GvAyvaQxDQM1Ecrh9Rb1LEYGPAuGte++hA0hS8N1kB9DZoi5sKA3YNR92LElzY0FkiLvURBkESxZbH//yFlUZohORpRQPu54SL0Uk+ff/6fP58z5Dx//o/6Hy6u2zJs5darFmSfZSKUbx/iLEqfsv3HhbhDHPq/EvODnmgHZdun11xIe7OSlxBWllFKvE8bv7C49PsLFWY/8cvPDxLOAvQhKTt/8xZT30EO1V3Ktk9QWUzdBdq1mOdQsv+Any5ifggPNwSnZPtUMI7iu7hL1qcC/QInzlGUUvM3AaT9/37+FoULuV9ijThHl2Er0U+ZKFmVHq9B9ONbK8Q9dfj4EkX8dfM/9A/DsUMTHOsB09THFgvuInojY4umFohDVkQvT2yNv/R5xLEvMU3/cSL8wvChGIG7NLVAHOIC3U1mG4yESgfa8a1FHwcqDImGmohDQBuMDqUkmCW/7oYOaOIMrAhVwDlArLt3o48vqkQ0aDVpoNHrwHX0sYZUE2oF+ON8y77ogQrt9hAvGGoCWk2+S/MpR8M+2DF26ccJmXuH7fYZf7S9HYn1nQFqpXynt44+do/jyzLhc50eqLQCAzX763a761vD1h344mCrqQY3OvfYPtiK2ccJOPxnPWbsuT47D5zzzNnb3r4RcOA87tHVm2xws+jj+pzZIU5Drw7YADgt5t5vt9dDGzjf9ZlkJRGPPo85GvbBt6PzkIfw6xzr2yx0mbu9vX09pMVKfdaPol0JRzterzG8CUYvZ1+ziOO32iA9bGjRwCKOP3WauL+t4T/ncNd38JNcTpzgPOiz3ceGFg05cYKp05af19RnxPGAE4J97OAd1Kfv3ulH7pBH0bSjjjga9iHfwHfYe8zZDIDDw0cfbn+4PWghJxJLysL0OV19fShPZmtrdMK9j+C6vfjl16jP+S4RrtB+IiCAbYhjH0NZn5XzCO3ziZqD8y219Qlxv4ovYGb8XhM4daHPm2oOZyGrvOBr2ccKIeHzVg9D31Xl9xjYh321R/p8N0QLfSDleNrrjCQcoc+JcU46kNI84n8jYd9+2Ar5DyeOe444EXEekz43BeczBYdEQx98gTcEU1rJYQ3JPr+9T/qINZLAcaNkPUlyjh/GnOL2kXFInxtqDs3v1ayHzKIP2/Hj+k5x/3nK8bD/Rvsk+mA82JXZh0RzfryME+uj5DydVzNX+2RwZtFHaZ/p65a8g93ej1LMf4jjEocLTuw/GZya/vwQK8B0ebVJfvp3EQ+EPl8q4wH29aJOoRPfiJOKO3vY/3yijjvs5772egwZR8Tr3xBH2v98Gc+Pt4+1YSvW/4S4T/cLe+P9D+UHE/E6CLXrIbn9qYzje/F107APfcRhwblCnIfUn/5VcBzihKlzlthL+vUqSR7yBPU5l5GHJN9Pw39keVWcv2XmVSQz5W9P88Q4fxN5ooqjaR9Z3ruG+XWS9xLHl38/rfECm87j2zReEA5KnOnTyB9sVLxdyH+Ye5Wx0xPjEgzXGeMSlqiio4/zgLEzE+MsCHAncsZZdKF17IMTGrsT40ZwoJt540Zd/5GNg8GBuk/Hwe5kGKV+Dvsgu70ftmL+IxvXD7evj43r3elx/VBfH9btuVinGHKqU/hUp/j6xFid4oOpOgWv6NtnhroLcZiuPvp1JORo+0+y+qVLV0fYQhyyRLxpTWVvyNGOB3SXksUdPqQi9D8n/kH/MBTfI5BxKL69ehQ2g/r1949k/StxUPT0EW7okrVt6mqWxKVsUbyxp3ofbl+O82sd+0jqlk523dLaHMxw/9T10Re4aG8D6idaW1eAYIfUaUZ0KMXB8QPNw9fxn8NUI479J2Q2aAIdHfpPwMh/6FBKMHvVro9G1NRciv7wiZgIPzpwAA61+myV4qxokBNC+ZuGfeD78iGFAGi/DkPlLEis3gSPAgLEN9j3JOfp6mNHNEYXWQ2mixvM2dp65gqMqEkT0Mqditdh3N5eRSnY/0QhNmmR3TYZBny8HOu+tQOWCTGKR/X0KcTRjdcOcgJLJAMew0FH7drS0o8Cji0A+lPg1CZPCuLvqJMfICek9GlA82lt9iKeHdrI6WM9O5r6xp74pZXvRINoxMHvydmKD7/CCl4y4IApuIpzHKWYPi3k9CiJGuKNA2b5b6M+nSpysEpvD+i4oT5d5PQpKYzoBpIVPIL90kd15GAvC5xAztGxz2m0z9WYQ0eCt4/t29f+5SpaZxV82A0Tu0+Kjj53kHOJkunooviyf8P9pTUKBTZxvPQ5yTpkDf+xAvDTQbVFnMt06OT99tFX269jg2b8Cu2n65a69WvLR05FcO7SoUPXYLf0ZzVntE5cwz4SzsH7YJ/9r6k5VBfTrY/6WOerdMf12cL95TN91gqtP5CVpuuWglPcf8ArgcO7Y2WCH7SPHz3aXr+HHPYv4kjqiZr6yDh/xP3LBTga9hEuk+K47V8wtn99Z4iIBwiLrqbPUdpHuEckGTtLOD8g+zyr5mB7k+ujxXHbR48stzP0YZQg6eozbR/yn5cD7OGAg+1+Jc0ZxQMdfaY4bnsfs/avZ3AS0dIHPyetD14V9l5Aoe0B7Sc5YVwPOd6GrWB7m+K47eNHwH8yOHaoXd+R6fMS7l/O4LSYqFfp2IfynQvpeHCM7QP7UFf6gKyU5uA1k9ff9DjCf9Qc7HaXNfNRaxM5F8fj9SHqf17zkPPkEnEa6XMGTL8+ehPzg29SHNH/dChF/D0qNcHBNJXagYZ9JJy4/8ngWKGifp3BiZAzEJxUfiA4NnG8KX0Eobg+Ig953x3jhPfB+9qvj+chE99toN/eZHnVHuyWmuq8Ctubrv+wDvppgzhDkSdCPnoM8lEXG1qNU36Q5ljQBvhHqI+PslmI00BOZyzv5T6OTp7pOUioW8Tx0+e0knqvRj66ghwvlcfTeMGzhYMSZ+IcW9XeMqSO/ULARTgI6eRVGP8cwPDWChssxJYweVIorpuOPjXgnEzGWbg4ssYcPDvgyOmwjk3D4UnRfn4VTmg8NTFu3PK33vMt5ISsCZz69Gm68Y3akiOKhyF98Q3GsQ7LGOQHjwO2CvmBZBwslMrUx07VUbCQtjoxrt87cGCNsfOURDvAUc1HyvYfN12O3qAfdCBSDvV7p93eQLpNdctwwn3EhDHSJ9N/mqf88ZMkdZfDW1uZdRfleDvFaTRS388J4AOTuuV52ODQpyfgEO/ROKFLh9LixfoImoLjrXjj5+jP5ys4Pp3gYB0HdSCrxUVKcUhVtxxxas+gOAU5M0go1lHq6aMtqGGB+SGdpjHHF+sos9tb863AjINC6xtrWyhXFBx3d16cbPs4t8wxC1l/ikLtQCc/mFGoXU/5T5oz1T3OKtn6rLb8OXGy41urE8yJk93eDobeHBjYb0/5T0q8YB4cXNiWE99MOXS7y2J5/jMXToH6m/l14/FzmLLtczAIzTkk2fqYt+ti9+fM/VSpz5zjTsLJ7n9MKcSp5PvPXDhiPfpLKD9W/JU3F05+ftAx5kBD+57v59nnnDkHwmjg5+lzZi6ct4ADjQE2Vf9zKjCF4DxvGHPn6OPJbodqCc7zxnuD2fbxJu9X6wrVr1Fy9HFCM87TecST/pPmWKYcnDtboD81o8TzyTEe5OQH8+As58cDcw7YR8z3X0IpVn+bQUbrCsrOr3GchZ1ltv9UTf0H4wGn+f6Z7a3e9U1BNP8Y7HMARdX/NB8GZgycp0qSbZ+3TPMqug8YsDz7nPQ9Q85OKB4xlq2PMYft+oxRvffAEmwq/zHn4P2591leezPnYB0TrZId3xpBYMg5z4qMF+onTTm7yfyDTP9xTF9YybE/xc/Ibm9ctVyxMAf9Bzkl59cF44ExZyRT9klzjOM1iCXm92bmB/OI19yFD6l9iHJDxTGN1yjLz/r58W0eHHrfVKZ9zONOwik7viWc2u+2YFPFN3NOK2S855eujxX1xbzo7PjmGXOS5wll69NNhhWzCvfjiZHZ/uPe8g05MA62CsxXNq1fI0fcX8i0j1S+cm7duufcax36KggO3brXusvvHnbuhkoOveduhnitxQH7xP6Doux/KoYcei5Ofjww5jDwH/Geu0z7dGWXTouD8QDfc5fjP8YcEHrPXW2bVnYq/qRpfN0SydZndW6cbPvY8+H4ufnbbWOOJzhT9kn7z+fGnA6z/Vx9JPerdTkNZmM/l5O/SaZhaHJWGBvI9EnL1LR6TQ7dL6n5ef4jFW0Ol+kz33gtxEf7XIPtTyqOrO4/n3iQ4kjvY8zEyfaflmzcqB1H7+Tqc1A2Dtbl8C9Ynv9I75vp5QcNRf0tJeYc/7DgZPuPOSeoFqknmnO8Slwf3b4Gm8p/OrKKrxanURHtINs+zallKbqcFch7sRPLtk99crqhNqda6H5jdWrZkC6nktxv/AnKTxUc6blaHF5l1mquPuYcGJRwvM+UHd8c4/bGeqxy0s+dz2fqPyjLR/w8fZqyOxkzcbL9p9Mw5XjPs8oPZfqk/0o2L02LE9aLzEfyqoYcen4vzUfKtI9XMeSMnndr32/DptTHmDOaf5CpT4fPi5Pd3hqy+5rz0Scl9Ylp9TNwLsX6vNGGTRmvTePO6P3oOeMfmWj5T/L8p7Lz6xhTuj6J2PdRPi2dU7Y+zUQf/fk7WpzDKn1SMof6TvzbeQPlRGmcQ0ERfaSL7rQ4jfh4tv9IVj3ocjYU+qQ4smG9Jif+qs4/UT5TcGRlJP1xfb4+8+OU7T/J8rOS6yEjTrZ9zDmJZNvHlt2nLaEe4sruO2txThXSx3jcaO3GC4+m7JOSjmkeYr2r8p+UeObjH7FAkdlvo5wtj3N7QfrEnGz/KVGfFMe4HYw4dnsdNwXHvF2/e7GIPuZ+GsUhP9t/zONOMlGi7Hg9+sZnSUrnlK1PKxC/y+5/4gXyZefX1u048bXPruNWFodfqC5EH27FflqyfUacRelTsv+o9Zkvx7oQp+jZ8c2YM3pAV9nx4Fw8hJqyz5zjQSKLqh84T1AkTw1Vix6nUL1qfpzS7VOonmjMwfdakTifkZTG6S9GH9ZS2SdftDj2YuIbS2ZkiKeOlOg/r4hfpesTz8iwz36LW3mcRcWDWGawz0wygz5aktSVnbNd3MrCWANV/W3OnKTuX7J9OBcPJpxRnwHznGCNVeyBvROFG/SIbwUniW/fkuhhrCHz3LDr1+yB8zB6OLT7qr8seP9HdfamFTY7D4PVKlvpsFubNWm9NsWZyT6c89D7WYCcRtO6wOtV9V+a2KdiXfG8F/zgFeCsAGdFWkdFGWtvXdx0OZc9fB7Sr6u03C+LY+Q/FcsHjuX/6rne6QBSdTXnaTyYxT7Eabjstts/E1bYIIOTSO36Nmyz6NNw371dr250KtawLq3bp2R2fTy2c5HVOs0qt2uy6YVCduIVubPbJ2CnKqzirVRtvvmN6i+tO0l9dFZ9LJ+dJs5Kxbogm/5Jwi/OPv4RHBufn+YLjq9sB6P5OzPrU7P809FVwbmqjgdVo/jGmbdiBWGlXm00GhXr/XzObPFtk3kNthNUqvVmp8EvVBUPtRznfHwdNk19sF/o9rt+xe67YcMaOsrl5NZFE32wn+v2oZ/joR002EDdz1m7Ju1NQyIT/9GQ5Dm7zl8+hu1maZxEiujzXwAAAP//7Z1Ba9NgGMff+EpSITbuIERW7Nhxp8hACxY7UD+AsLLToLIvsMtwB2lTBlaG+CF2Gg6GXt3BjBy8DG87m+Fthy7iwcpq4vum69YtSZt1Sa3x/8u2prD2t2dP/nmgkDdxfCXdny6jqkfZ4aSoP4dNth0l7kF/hiO7zUlRfo532Jai/jQ5yM+lPegPPAT9GXdPQH8kfbXWaK2urkqtWoPtSPxHjdi2q9gue2Ao3hNbOWA4gnOXIRw4+QOHPbSLxZJRLJmm2absu0jNdsnUA+qBJ5LniG8pqiddnqzDSU89qfN48UlRPSnzID/wwAPPqD3SiDzEDzzwwAMPPPDAAw888MADDzzwwAMPPPDAAw888MADDzzwwJM+DwBREPQq0SQrTyh1qOXaRcEefB3lUB6XaIpdMiTqSLZru7SdiOfmB1O3c4VlSxGJXCDPzUb2vpGAR/ler9tazqowj5oju/W3Yne1pVihJvn8XpONyiTzyMzzhiqDXzWcRyMyqTwUiUaEelIecYkY3GPMiq1ZS9BNmd7RE/Bce8w9qqIvKe0HNiVVmd5IQMMXdfM8xresWCxQ4mbDbncdh0cjFZNIhZworDUSac+Jp0LurRGqySKtm8cJegwy63lkSnZ/JOehOpl1jY7HCFqdPyaPxA5rd6/j2Uvk9MYX99M1mVjLNCuqqkrJl6Q8pq6ppGJRMZsrqMLuq9DLkK8ImwuldsmgtK3YKnHDl424IlXuYXNOsKmlkqpw5btaA5A0eTchjL/jubjGwHXOk17m58t9WVhY8BbfqtUu4+kPv0v49AkzMzPvfGxvN5vNMI9wykQvzzj9aymX9/e9pQV/X/b/1gdd11932fSXwtja4pdpRvXMcc7689SjT0krK53V0X7G1x/G1NTUSYM2Njb8JR3y68wYAZ5bJ5xrzsRtzqDulBcXF72VH7/G1p9MJnPanfX19cD+eBfRformuRig+fmBAXoRe35IT36mw/LjOGGe4PxMRIhPNz/+AA1dj96Tn83NwAB5+TmO6Jkj5+LTCVDfmpLIz1l8WIACSurm58jnOY3PraHjw/LjC9CQ9WQyZwFaD8vPx+j5wfzB/IkE5k+wB/MH8ycCmD/BHswfzJ9IYP4EezB//sv5k/cdkDGRcs+oGFU9o/JMWi+Vuv1IMlp52tlVdlslyWrn1+xq6G7v74ftwhOHJ+d7k/BXnu0O/lN+wfNPedJ2XMMz3p605QcenHfgGX9P2vIDD8478Iy/J235gQfnnVF6RvV5Vdo8AAAAAAAAAAAAAAAAMD78AaXLy9M=:58B5
^PQ1,0,1,Y^XZ';
	label300 : STRING(25000) := '^XA~TA000~JSN^LT0^MNM^MTD^PON^PMN^LH0,0^JMA^PR6,6~SD15^JUS^LRN^CI0^XZ
^XA
^MMT
^PW1200
^LL1800
^LS0
^FO0,0^GFA,277248,277248,00152,:Z64:
eJzsnM2SnSoQx7Gsum5uxW1W8UVS5WvNKphVXos3uK9g3sClC+twhQaksUFnJmfSJvZiRjnY/DzAXz76KMRtt91222233Xbbbbfddtttt91222233XbbbQVrht9NQBtXrm783QS0neTq9WrDU0mwyflUNp5ctQZTz6YJVunHiVxMuTxWAJOIsrVn4XvvIevkThsd2egzdVRiZM2ZVsOVa3Ox2PMKlwwgjyS3/zQmWI1MnURq3Swp3EtwtakHx6UQV6jHMtdCptrMzeZDyLE7FAqmXDXycMhVx0XtCVx6mqpsWmgLlR6aI6HgytXuHBS5fPYlwwXpck9bzaIZ3UUrVHUkFFy5dg68VPoMr+OC20m5Vmf1KCrPZRr9kVAw5cLN3haXcMGZ99InXDuCiUxVov6hxxd/0eqt26vtFbiaxMERV3wDJMGSof3UDC9fvJNhLcV7uBZXt/vCi1yh2rNc5rpql7gYri+Oq37YPEWu1O90kktnrrd3tufS4t9m+Oy42lm8vAipLsi18zD5ql1wjsG5TLgIgonm+tr8nN0sux+r+Vu5Q16Gaylz9W/lUl8bPTqudTQxy6EtdUiuXKl8/QKuhfBquX4MwFVrO76vS0Lxp3BFBb2Oa/rUfB9BJ9YKlLOcRWl+z5ULGMzI2x1pL5V4Qu1G49Ho4+1c/VTpWT7W/5flMoXIt3ARBDrHNbx8s9dotU4lpS4KBW+uJSqiyBVNnhCXPZGBq/MHW0Uv9Y/h5QXubf185SoKBW+ueFmiyNVnuOBTibnQ6tBS+fmQkQnDNZWEgitXzADH6XS7y3BNe65QfTGXc7uIdWQzWB8rkOFaSkLBm0sdcrnp9oaFFm4cQYBEqf7Er+doVVsuLQpCcREu86/AFU/Oj7kmzFXB3GVVhxa4VEEoeHOh9nfI9fOQC3lFWaxM9MBVEorrcfnTmKv9BVxWJixXSSh4c6H2lywDxGX09vh7VBAiOMVlZcJylYSCOZf6MC6QCeAqCAVzrnjzocAFeasjLqw0mAtkArgKQsGcK9rqSrjizUg4nrNcHcklERfIBHAVhIIrl3MVg4Wk2NR5roXk8gAgE8BVEAr2XPRePuaCGp6iBxVdYygV75Y7mdCjzZsXCv5cASzP1ZW5/IwMP/k7xOVkQg8dJOZ2IblyxSsc4zkuleMKBLHSVLEDYRbHzdkD8qyQoyCNKxdaV4MkmeWS7lCSXP4WJ3SzyMHqwsmEu9JsyVyXi97LTyHiyR1NkOeqvEz8A05UnQmj4MqFKdQJruVtXFBa42WiORIKrlxdfDG9N+3dNue4aKVxpXmZ6EYnFLkwCq5cOH5ClbiguOmAayG5/Brd6GRCutGSyMWBceXC8Tn0nqZzS3DRBEQqPLYrPYBMmPhV60Vl48C4crWJ0zxXwJGhKJqASFW2rBWiN2dDE0Y62Tgwrly4Igtc2zO6yKXIngNcayO3Z4ZpbMFxNg6sxdcfcYky1yJILijKdUdtcszuMNshuXLFmxiZwVMU3reIqGMSXBPJhbvjYm7x4ao0HzDKlQvvYmS5OoJrTyDIVGXLWRHspZMtY+jN37EQMMqVC0W6Z7kkQbgjmAQdLWdtbeL2AmUdgFDMpYBRrlx15OF9XILkcpNtObpBhL1ssqU+CkLBliuCoafbE5oq5rnijfLNXDVW9rloTnX0rxjxzpVrA0uWjzeahuDaESiSa3BleJlwzQYEvSgUbLlC9R1xbUZxUfUYqinIhBspqGOh4MvlnWW5Op1ajstXU2pBJnqX+YRQsOXy5UYPZcwl81zrp250uRS4Epk4KRRsufyiaI+4tqVSiitaSD3mSmXipFDw4qp2m/kZLmI6grhq8jC2VCaKQsGTS4bvfpuGZbiI4U+OK6pSVFgiEwWhYM2l38qlYq5oE4Tm2slEJBRp3itw+TJ8mWCdL6M7x6WyXPVOJiKhuBSXOsMlKa6I4JCr3clEJBQK570CV/c+rmga14aj2PqdTERCkWTmzYUj32guarVuynD1JNdeJvJCwZsrbrf+Mp+jc2VQqwMU15LjomQiCEUaRsGbK965mJJBiixyxQRdmctG3WssE5tQJHFgzLn0Eo5yXPjX+me4RszVT3uZ2IQiiQPjytXty8pw9bucKdf2DNcUl/nRkE5kYhOKJA7sOlzqFVzLK7hqTcmEX9JMhYIr1773uwbuZ+Zh9OJJ4lT8zNrW7SguLxNj0oFgyTwVistwLRku9+1PBa5tYEhxeZmAzZfNJtcbsFBw5SJWtN/P5fIOiMu5eCSvLYEtP50GsnLlIvYFaC6/UosuS8aQ0nmguHzY6pzIhBeKNJCVK1eX5kreSoMXBxK19XOU4ZjLh62mMhEFsqo4P1euRCiWlAsv1qVcmEA6FxRXP20BHdjGMwLGhisRiinHBf/CejbJ1Tku3HPAgkzIlGs+I2BsuJKGLzJc9Tu5gkzsp8cPWihQAzNVDEcjyRWWQQtc6YjEWuiOvrh5k84THZIRF6pwseOCspYWp/qL/kMEvi0SXGl3HKP7oDskW67ogTVmufpXcKl+z5V2R5dqLdMhuXJtM+lRPMtSmVBxyRmhYMvla/J5WKlMwG7A6CsyCMVwDa7nW4dlYoLuNPiFHy8U480FJrFMhPfx1Vgozr3q+s/nqrBMrCOh0SR3btUjCMWZV13/DVwNlolJ9Da59qtqv0souHIlMqFqHyXmGj7wTodviv1buEJ5TiZaJWBU5Bq+14dyHBgDLmrT55fbsO3G2npcxFdhatFC9DFX4OfKJT+Ca9zeTOvatw22BpgeyMHCAVOuD6lG+xNfaN8QEKDqtdk3ru7M88n9ZnqqkwkMO67+Q7geZpzTA6HURiZMNboqq0OyVmGcw5XrQ7BAKFog7AzXKhNVUHbtq1dv42imXLul9CfZuM7ToCwTcbIYmeiGiCvEoQy8uagt/mfYbNYBgLAycrByffNYa9/b4lDEM7n+BwAA///snT1u5DYUxykwsFJ4l+0kMEZXcKpsYayu4iAX2HQpghUNXyRHIeAyxV5BQYotI2AbFYKU90FKpDReYx17hgO8f+OxLFE/z5B/Pn7ozctw4TV0kS3GAqeIsEX3YHQK3tehxErbTBiQ9OXUgxliBPwWbBHvAAU4rLJWGajXHaUBbOCmPM7v4c/4kg5Pi1F0aKttxDXbxJA5V01nwg/6o/pY4AtcObPYc8BYYaBvKKloouN9MbVQW03ggsJoJq3B0zXUa9cggMEVAOKy9OnRlk0Y8C9G4aAIM1d7gJ9tosuci99ZngRqmYs+nFEtXC1xdcy1VzHXQBDEpWYurNSIW400G8f7hBOjQK5aRVyzTbhz4Cp74nLV+LEYNXHBcP3vwGWrEbnM9B6i3H0xfYIajHnJPJcZkauBroW4oIQODmJ7gUIegKuYPidGUVI3FM3w6jCqXaYxv8L1T8RVP5frr+dxccKFctC40kSl4uIzHIaLxwauhfJxSuMzT33bxv5OY6uIi1u/hTAGCTDBmwUqjVxQyDCpwc8vzUZRIZfuEq6VTXyVa1q4/n0u1/g/ubobw6X2ZhoMcOEb67m4DR/iqp/g4kJ8dQ9GAUeh29Zu4VI+49ZiE+fD1dbERW8sFAlcfTlzQa3vI65d3V1HXO5Gp1yhEK7uwSjaCsMcozZckU2cBVeJpdqUSy9chrmKNZd5iovrQReMgrluUi78xCP7ypWrDlxQ5sBc6KCK03J6rorL1RT80GakmMs/59843tfjuchXuRC/+2YIRtGCuzjVbbkWmzgDrom5cGaxqx17A3C5oWw9F0VCwGUWLtNBl0O3hX4o5qJ+yBcy+bkG5Y3CNhgWJlwNO8qyipw5V2+e5sIVk5FiPeLCOGdvHADQbTECpJlw6rc5Ltx7LueDZG8UxJXYKnNFNpE5F0RmDiAiLowAFcQTukMungSC6olcLUZEERdnNMX1OuaiuBAhkauFTzEs6eHRInAltspcfbSIHLigb1u4XMx1M3M5ONvyGCfhcj6+551YPr6PuXzaCGqQzWEubPNttBkgcy6Kwmf/eoQLPyZ0cObC9ljdPwAXjf2wPZKd0/gROk1uj8Tlo3dqkBVzpXbPXDbabJI3V4m7ktwQ+kdwbuDCW0E3d4ntkbtI6AmRC4x/5tLoSLbi/pG5sOHMXBNx+TVHbJDlo1xjvJkpdy56UqT08Re8ru4Wrj5wdcw1rLnaLVcX+kfiGueIYiw8V7fhim0iWy4Tc4X4HrkAYOYqn8sFZ8dcaBRU7kGuNn5uLlcuveXSCRcEA1/hcuZbuNAo4NxDXHi46s6HC+f6jJ9dgPtSEBG4oNRv5prHjwkXGAWUhFxpOIFcY/Lc73lw0XyOYq7Cc2Euxgq5vkzUD42NMwnXlzHth2KugrjqsGOVjQK5HjZcffJcea5cKuZqeb7wBrlw7cZz0b4j2g+IXBhEhjinchCxuzBfuOLyS/s4yREWOfHJYdsc5mrTx35z54IoGJdKgcvByHuiLCiBqw9cE3PNcXTVERfH0TrmmrSfj2auagpGAQRgCPqTWnPZqj8Hrpq5HHL59Q5FXCOtd2h6Rgsn6nlPPdqtnhKuge5K+wQjLqYZab3DeZvA/w2a0EGu/WpjTs5cx1OHLo3zORuu3SqvT65cx1p/ZJFR3ALXahs0HFzljcqV61jr2160X+kQ13o/Wq5cx9o/4YVGgVubbjZc632FuXLVR+VCo1C8nhZXJpyusefBVR2Va+DMUVuuTdq7XLmKpwt7QeEsFEbXl2uutU1ky3XkDxJcFUYYLuUyh7Lx5cp1bJXbjFrIZU/BEitXLhg5N6t0P3VbHPuxjq1y5cKv/F095QhcR3+caatcufYbLhggtidBSZQrV2lNGkZr/Cai07DEypWr+FOvudTFiVhiFTZPLtXqNA2AGdSPJ0JJdLvl2p0IJdHvKs2Ht0oKcDLlysW7KxZtslWeTLlymXRtw52KY61cuRKUVa90UsVVqh4eP+/YypUrZsmnOebLZZaKb/Jpjvly6Sna4nhKkJVy5VJz2jWdU7XPl8sEnDqnap8vl554wl5PGfVCKl8uehaTZsOzqvb5ci3fp5OXcuUKC3nu1Bxr5crFK8WZuQQqVy5cyctg2n6jXLlUmSdWtlwikUgkEolEIpFIJBKJRCKRSCQSiUQikUgkEolEIpFIJBKJRCKRSCQSiUQikUgkEolEIpHoUfEj6PVEuYEL+E0rdY3f0RhOKPll2SpX2VoVd5MdqlG3pXtNLEoduwtc5TRzzSlSPZfplatd4/TddDdWo+mrV01xoUviUpxL+a22+AO43Ltwhk8aeXWl3Ye2deU9XvPd1e7du21pL6cLJJm5doULXHPOZ8+1uyyd+83dvrnHa77fXX541ayNF0XMda1uH+faO/eTJa7C7naXt5fb0l5OUPhl3yBHr1sA+sU+FN31Ffz+833rbn99j1x/7C7U9cWVQ+4f7vGa61fnGtSb/wAAAP//7N3NjutGegbgqimja5G26OwaGVm8BRlepINhxFxKG7OdhYxZmIY1LfYImM4qvoNJLiHZZWEg1ehgzmYwZ5vFYFwNA/EmGNeBF4dBCDHv+xWpn/45R7LUHifDMny6m5LIR2TVV18VKbGm690aNftCfVDe2no8hiv/vHL+p3O4dHN6CpeCS7sPfjnDa8anZ8/renepkgGPYzIYDqNrcDpGTDg/Hw4v/O1teaLM4ldn0XWRlB9dN3jNhQ3P60qsGpzQhX9Po+v05AOnmsBD9U+3V6VtFnox7lzuo2vzucUv1XT4nC5EhlMj9f4EWxbXmfqwRPwaj08++udbDdev1G3rcsrflPp3pnTD4Xn29rV/93KqV6582bn+Gn8P4frgXxYax/FE3Xhxoe1+fFWq3+rSnQ3S//reXXmp3Aldf9m6nBMXuoIPNV1X5fgk+e335BqrGCfO1N+46Prxj83W/kLI+BC9UnSpZ63372y7zug6YXvccqF+nQ1wbHX5YfOf6t/FdfG88d607fH0BMFzmN5c3Z4Oxhd0nZ3+1V+Iy+hfwnWqHMLXVF/r3xijxoPn7YesbePX6Qni18Be3d4Ohoyrw/FwOBhEF+MXHnUXynu9WFxbgz/Px8/pMkv1bp2KC/HeNm55a6vxOeNEUrUuiffMc5owd8i/zNLgz9Q/p0tV6jQk4jIB2ViYxf4RcdX4d94Rl/SP1tOVKl3WqjLKeN567lnLVrt61oOzX3nW9n5A6V37lR+qqy99eb5y2f5Mm2YQfzMyNeAxlFXxzu3rknR/csLgQjUKfYSamsbzzsm1rtTxOoH4RZ/jDVf8BvHOtfUNjSsX7+XAGyfw5vHB8Cbyidwa9Ghfuq/jVx1ON1xyo9C1q3zMZXnTEtvwxr064Ge+xEO2UfNj3fnFIBUVlxqo1jWxPv5Cl9+6h/BgBbQleu6rMEnoUipDSnKGhcWxBiO2DPddRXf7FnHpR10j46wfqOk5fHQV+H+MhWGgjlMsSduu0N2WWlzKP+Yaapf6oSoKU1q6gi3VBRb6Z3R5VezimsB1PoVranm4S+WH+sYd61YmdA1yNi+4Jmz3OHDnAyTM1g1Rt+D6uZtrDDlepCVdurblkK4ZwOfKlIPpQFoJn3Pj7DFd80V0NSWy5c6VhiEODlyfuOaKrrmjC0l0eQ6Qn7auEV2ON4I5qgv1ftB8Ja6kcWj3OCIZXfNqmMhxhPrOTfQLjBwHDBVXrqDr78Rl1XA6uNS3gUJzPBfjRHLjpX4lty4b0TWkq8iGI2mPMzzHT8z1XXTZKzz7PFY8hD3UMVBf1hDioaO55E7EZYgu7dHeO1cYDhGMUM0K7FO6uGclQgS/dtWqgOvmyyVcttFHc7EfStQ0ulBp1i4/GhbSD2HZ1H8C15Tf540a//HKxTuhTaepuatGeL1Zap8cicV7ayR4zzFOeLT31nXnB8Mg/dCUj39i2ULgyrT/zLUuzZso+ulQ3SGGsX4qnx7JZW94dM4fcTn1vqfLTfn4zzsXRHnZuhBHpLapVx71X6XWVfmxXIwTaxd2z9rFEbU3Xlw/vY7PpCjtXIgj5srhtR87E4Pa/PWRXDhGT7uCxAm6zr/6hw2Xal2oTPq2bF3nCoc4//pILmzzSddoStdUXHcbrqRzIY7oF2sXH7p+HpdXXbyHi+2xc908tr9mdPHrcVcudaw48Zjrvc6VrVzv3/x+7UK9P+MUMPOO6JrCFYPtsfKJ6FrFCWY4fliIixP64kIdXLtQiX7iWMURvPAgXUPEt+jCi47mKlZxFRrkLSrkYaARVwfSD+ExiN53/9G6GFdbF8JEgf8Rv5B94NFzfTyXRKW2H4KLeWeRBPRI7Idivz1FP/RuWbUu9EOvPP9FF4V4gfcx5fvBeyPWH+tkA+Mq+u2idWWJ5Pf2Wvpt5jmIX+i3k5WL/XZgfq+Ym/L508S4YoR3gLgaZkdyYYzF/GbeuvIlx0PBLiXPwc5gvOc4rAydq2Ek5VjOJ02V4ucUg6O8ZjhryqONh5hPIB/MWxfHgxwJ1t7ngfkq+0f07VZ67zYvdOdy42WfNhWfDzdvLOx5Fjr3R3Ip7qkJ0qjo4vhZ15eq8j5BjuoVosAUY/K1S1e2zGS8TZeMt5HsWOnG6yOOt5V6GHOe9UzZ7uWB650/heJhOVbMOXbpXfuV3tWXP7uCvnne/T5vms+7xdIBIwGTSad7t5LQzerysNRxDY1cR2Y5BWoCb86ExQeO2EzZTrHqctOVNluu7RvObLjmnDDB4JgzVQldaU0XFh94jxpbmvaCuC3XXFa7dvnN12y4mgovtI1HroPOP0dm0tDVVHr7JXuXBGsND11xy2vX1vz32qUb5BAlhuG8H6C45nRdIVU68JZRacmUNbrgaOc9dG271dIV9LbLr35DgpqW6VWVXrNGYQBVYzRusdj6w1LEeYkc+aFrLRGX2trI2mX8BGsYqdnIeLQfuJCeqQEWW3fYlHlTJnGed8uFrXSS6CqecLkR1jBRs4mOLh0sRktYnJQHuczr6LK+deEwLLk9FUcQedm5zmPoUNguXfE4A4A1ZCrLmNviNZqjt4yuw7JL87W4zMsqr8Q19wZNC8gZ8mXsDF8gN4ZrNEuWtnzPvPjHIK605h6h6+vyVGWnMhdWxF1ZiGt0kOsatQPr/7JuXRgMoWnBldGlm1BgD9JVp424/q2SjedL62a8ezvWoHgAvfmGLicuPznQ9SMbXfWkdd2FZCEzWxO6zF1V5HIKJP37SXJdnpsXIbpmqXGMXcmPrLiMo6syt0Ga7+xAl2pdYdTWL1claIqo/iNxuaK4lA2l2IELd44R70xcRWK8uKTBFKh29qX6bGlecqSEcHssV9K6Sgyd1y5bzopaomyKo3PrMnuN9o+4inHu1V1YuSo0kORzPM98uSQ790dy+c6FmsQpi5Ur+7SS/nEkrp/Z63Ll+tZ3LuzhSyWuRdOwjs1DguhxDJe97lyZTPFEV6LGn4XWFfSd/1lio+sK8eB/Vi4Mb+cuTVSd3FZpyWE6wuvlW7e9g8s95VJzL/1jdP1x0zV3ncsiqLIJjlHtkQg46YcOu83WQ1eOHGHT5aTeR9dvostL/JyXnQshTvPcrTJfeTSAkmHtwNt/7eZiraPrxaYrX7kQ4hRDg9JfOayqtA6R7w/P7PJ0zejyr16MNl2qczE3LarOlcji5tdHdmWyNMZ7bOoXDJQqi67FpitduXjICiZpG67JUeLE065PN1zfLn792P7S1SOuA2eFbOy3H7jGrWtcVGvXZ4svtus98xxeEqBOW9edi4sS9k1Hca3i6kRd4O+siK6smG249KMu64Ggi02jdSXHcW3F+wp/51XXD2VtvUf2snbxygTkHS3CqYliYwnmxrNiWAbZg11ldc+F4xESbHgGV4H9F+MEXD/R/7p2sR9iHi0HLXaqeAo6oBG5tizetum3uDjuWOcTSBTQ22HcgQBZj6yripRxtRqxIUxU1bnwtFdexh3cQSpd0DXDe0zpCpf25rBxh5Vxmqkm/PxUdN166XnMXY38KxRJGfuhSbLpQv6FfILjNFumTZ1wvj2O05gkHj5Oi+Na09S2al3MV7GFyjRfIGr7lQtD8BGrVdbmqzhm7bg257VMTlxYzorFV/sDXZwHMF8G07mY3wOx1A3ze1dYF/OJZImQNO1caY1jLPMA4jJy/h5PSWu65kEfPA/AeRPzwunOJdHb1LmawZUzWedVASNOpWy4LCr4TOZNxMUXJcx3ME7KZPH8bVvepWxd5RXLYd3Ikcojrh99/4qH5RHXD6L0rv1K79qv/FBdffl/XZJn/Yz2m8tUqY1rxudNU68T4HkcM8ukqxAfuaN9ujm5nzsZB+EH0yZeq4Y0LHWmQT6EhWaPXHGqbLex9+65dHuV+6brwZq3XEwGh3gdMHxLmbganpqpuDDZY24gcO4y/jq+5zLt7tl0Pbil/abL8OFMfuTM4mb4ESR5ZaLYLtytIJlPu50Q7rls++G4TdeDd7ztWhLDW6bLiRxKAv6ia7Vwt4JULtdrF6fBV67E23XFl9+qh+ne5hWY1l8Sk7hLVSdyoUfWLlTTxM3V0vr7L3+qWE71zR53paVeV6fW9eBC0M0FSZkSk5ap5sfno4sLeTUPflR65wae8pxB9oRLqYeu8k0u/GdrpuPag2DElcr1kQ4/rlaX9r+95Dz3M3nclXdfm7HhSt7kSnlyrcbqONceSCziwjgwv/Jq58Huku9h9LhrorojvKOLkwL5F1iBXfAkSfIFHROZ6eTswIIXMO9WdN255HRLdKVtWJytPl6EgLhy4QB1gXjeuZq1a57RVYqLU7XxbVo+tnC7u6qAsAXXKA/8FhFxzduwCBfPkxUJr0OTM390fY1w5DI8WLxis6cLC1LuFbouM3Uqc/pYydqV7OuSSzDpmted62/XYbFz4c+ABiaub2pevk3XtwzIdPGEbYkjzAm+bl4PrknGvZzFPYlqtnA7T/LosnM1y86VIwJKpF+7EBB5YlHiBK/eqyZ4sHrNgExXyvn6NJ4mumhdeOEsU6/qWNWHDBdmd1esz2zNYb5yeYZFUag0upaJD6zx6H3V8iy/qkeoeaG5al1YYN0kumTTSTy1mqnXTVmgurLKufw7uVBD2nqflxPdHrXOhSgZCKjAYRyYjTDwD0uGES7GAuOzbRfbUcb9XqC6cuoP3dG+Lk40oH50LpUaH2t56+Lp7sAgx367wtMnqVpqX8sL5fUTzoStXQj7DRouXf5TduYFFlTab8SdXVyVXBfQuRAWjQSNtQtMuTSVeU6FjYwS9UftK9nRDc/TjlSoNlwTfmEQdqGuTfiMnTmCf8Ne6EE68iaXlmb1Rpdy3O6m65t7ripsuGa8ANW6DP1rNefVsYFJhq70Xi7WpVTJPFuM95xsLTZcHMa9CirmOey4Unv1DZ/futhMf7HpquDynJK6UMWc/b9XMZ/YyxWnMN/i+tarmOewg0i2XZxb5SW1nUvLQYiXKhSX7CM8k4xy3nyxjyt56JKEecv1OrrSsnW97FyyjkRS+85lpNKmsusyzgzTBV7e7NUeueq3uprYQJLoMjcv+EGnDRcToM4l38FVTDqXccZJ950u93JNdnJV4rIuum7vu5INlyQds1l0FdEllwyEvVyzJ1yrfoiu5ezNrs39JTlGNpfOTFw29p37nDSK8eBhvVf3XHW26dJfXX+unqxfkyddu58ECbGWvtVVTbZdi5f3XD7mX3KxFT8R2bnOv6vLenHZB67LDddF2z/yWWiV+uvF79YuiV9rF6Kpia5bd4BLLprfiPeZxPsLHo7prIv3Bb8FpXUxvL9e/GHt4oL/DisXDoDhqT9e2MTzmdbJ6Uh+1nL3iYAQa+kDV8VxR0FXRVfV5jlJ5zLbLh2qdoiRtZdiMVUFrxh2Z9w47th9IibEWop8Qm24fOwza/S1Wq7YCW1eyPiF9EF9on+/djGf4GdXOE7jy+UKlEo+bKQqXlwTXWXYffzIc57iWudfWDHyL7rKHCpTJRyQBqn8Eu+ZrM7RBa9ckn/N2iFsxkVahrAZE6QkjiDZD3Gwu7tLjnkaLuWX6FK19ZwHSJCZJHBhAN9miuwfkZ5uu7p8VYb8mRyApZV+HOthhz3iynKZHNjdJZMhKbK3bjwElzRxWyU8Z9Xm91ou1GEnzYmWia7Wri6/t3E+J+eVtZxNyfhCTpiMlNpz3gTjL3GNmjgn0rrmHA8ZnuKfL9vxkApdnsOJKZ7QXrnieGg1z4QAgS7aRWLJhSOl9pxnWrmQhc/LlUuuQ9ZMm9O6HT+qKuaFQT6Uu+WS8SPbaxM6l6wgk/U0ceDcTdbt6UrjZTatS8bb2FdzZQNcpo7tg4c3yPB6JHlY1xc2TBecajsjuuRbPzKZucRCuvacx2zLo6cbk5CXe6/puOWJ06DH+jz2dy5PuMz3q3hYfhCnjR8pvWu/0rv2K72rL33pS1/60pe+9KUvfenLn00xzZ+mvG2qqXf1rt7Vu3pX7+pdvat39a7e1bt6V+/qXb2rd/Wu3tW7elfv6l29q3f1rt7Vu/7vuP4XAAD//+zaTWrCQBjG8QkDGaFBt12IvUZXepUeobt2l4FuPJZHSW8gdONCtJmP2sQiNBQ6z+L/CMlMyOLHi3mdDOLChQsXLly4cOHChQsXLly4cOHChQsXLly4cOHChQsXLly4cOHChQsXLly4cOHChQsXLly4cOHChQsXLly4cOHChQsXLly4cOHChQsXLly4cOHChYsQQgghhBBCSKl8vyH60pRRcE2L9dcDjeCaFlzT0nPS582XpowiXK+rgUaUXItIaONRybV578IPUBfGSq7242CMa57DWMm1fzkaU9f3Yazk6tZLYxrbhLH1OeX7V9WtVgNXvlq+XtVuOcf1+2i7arcMEzmXmz+GiZRr3T+P9ijXV2P/MoenMBbqX6nf5yjVK/4+5ii54noiR8m1GBDs1szi587fur1IlOo1DK5pUepfw+jW63qgETVXlTcI7XaWItK/Li6fL4jUy9g6nfzX3N+6839T23iSczWVDyeh/pX2xC+ufLV8vXBNzGtY3tcJorT+6lx/cC6OhepV7QLJnuJEyhUN6d1Dz5Ui1L+yS+55rDpNV/889gaX/uyr5Do89IdFdgmtv9rQIgT7/SZsmwi63N5IuoYR6l+jSNVr1O9/XisWUVd7HuxjCvWv81lyf7V/pT1dJkquneb3S3z9lfLXen0CAAD//+ydT2/cWhXA762rmkVe3Cye9BYlfiq7suAhFhQR6i7y1vCkjrJB5H2EvgVSkErsUqREBcFH4KlsqqlEv8ATcVWJbpDYkB0SjooUqQuYSlRvGk3G3PPP45mMnRnbNGfRM83M9dzU/uX4+Nx7zz2+/j/80zafJqKbS5H/YtGtr4S33nPVS0CNkSL/RVJw8bYWfWk9j9q5VPmvVXhTqK/3XMvJalHykn16qfBfZa7ZwkXKe67lZHXSDunxXzRO09c+8vhR3fwjc2mcfwS757gcu6/kN8mFEpGUuBL+Spu+Ev7qPVeNAJfMP6rxX4b9KpbU6StQN/9o9LaPE/H2WVT4r4no05e+eWRsHxXOuyOX/33cUOS/iOvK93BDkb6MWXc/K99NoKiKC/I6tHNp8l+gG4360sy1qvB6BIYrhf+ilwb7gnwT7xYWVekLbliwePuQJi7n7ycbqrgm07Wa/JctTW9r0teUeMnHBl/quGYLOkSRfZlgMClr0lek1O7jsp9IZgsXJ2//Nilrsq+jF/AeYVmRvuzRC2DIU9jwviT3Zb6VXCQTiH32PIGskww2NOkLuTzzCWwosi/i8o229RSI64pSrhV1848W/YRw6bEvcwR+VZ++zBeYt81cX35McvH+y3wB7fYHiTp9rUE/R7gU2RdKoM++UALxX5cMvrRw+Ubbuhgkgbr2keQDdf0Jko+k/6XHf6F8pK6/OiXq7ItFrb5+Re5LDZen9H53X9YHUGZfPGWrSV+W+l8omvxXAC5VuBIzU7g4CWGJQOFSZF+37EClvnbci9O/nP+6RKKAa2A2JP1Llb4ycw2MH0EU2ZfNYCI5UOfvbVrOg9Hjv6a5ktnChck0lyL7+qtSff2D8tJ+CxuK/Jcd0vVIXAl/e/FcZmiuFWVF9kX+nkWXvnaKsvfoOokC/zWG/oS+vDTvn9D/krw0Pfbl7UF/Vd/6OR7272WdLUX+C9+1rj8hXHrsi0S7vvT4L5JVffqKoAvt8/WoyL5i4PL2sKxJX7iOm/01lr1Hl67j6+Lty5bSTTTpy43TJqLIvty4YyLt9RXkrP9JvlssDw2qq6vgkvvmWvuvWA4Z5DQlAM80Gpxfdw6X4DTVFzxYKWUIfn5wKAu71NVVcZnP6b+2tS+nCdKAzeWQsTz9qa5ujmT4/glxyS811VeU83I8vjyMCiDo4SB1dXPkc3zn/NW29oXPxoJCKIf0iydC19XNESK6R1yC01Bf1h0lRFVEuf8Az1qQP8tQTTY/7W2jgUX5HuEgYIWB8RK6/yaclvblu+N6eGw4bjxEiIxSd/38Vf8JqgkVNzJ0ZstpvWe57F+IS3Aa6gtvJ4sHsNdUtl5n9iUcIsh7vR7ViZrimkeiEZf/gHBa2lc45DcPtIBv7jTaDCjDk36/fzA08pA2w4pj3zFfOup/RZl780f0446buD/bOi74Pnrj9LU1YmvPsS6vuyBBVgxxtbSvODUbOBbFuChZm8OycAXEr5y+nmDdHhh+Koqr8vgg32AuwWmoL3dyNpwa3Ek7Bq6DzPhvges/7vSBefV6UIdcULfwY+Vb2hcMRTfw2U8RJC36vx+Y4DVwvRy5uj6I02OEXFCXF1fmnH3l+e8mXMlsYSnxRsgVJSbeA669gQmPgOto5Op6d9zLnekYufaG5L6qHNg012OWJ824uDV2x5btELAyp0jvBPV1kLJ3AA985D6OFuJKZgtLiU8mHGSGjmVH7gpFrtz4b9C+tjP2Du70RcRV4Vin/uB29uWA8GNgyWacmmLmSoJXqK+nA/YOTk0xc51/rJb6Yi5fuEyZi/S11Yyrnf9yhoV7GYKhwe0/sRkjVhamIenrydAjs3enT57NmZ7PlcwWluOi/2WH3oC4IjMiriAND1FfvYLr4ByuqfsC2tlXxFwjX7juC1cW9UlfI1+47gtXNn9n3d0XEPHnyM+IK7w/JC4/i0hdvYLrD+dw4X0BMu5o579i/hzzBWDC52/J7o8HMemrPw4E57kU5jeQvO5wF+OhXfkMUioEz18T18tBzPraXZQrg5DvygrlPbazrzqu3SX1ZXH9aOESnGb6KkbRoXAdC9cwZ33FoeAcS2Fuh4LWoRSuh/v0aua/Rjils2GiMMHFshP/mLAyOxyzvg7CPTb8ZbgEp5m+6rhOC3014WplX7bgOhCuXLhOC30dCFchcztgHerLDpkrPDDE5U24Tu9g/+vO9qJcU3bfyn9ZOSGOi8TD0RC8Tk8KfeUlwZZ7fod1EJju9FXNJfa1vSjXPVwfYJWeG9jOvjrV1wYQra53cN9Jt/pauerervwQna73kKWR/ypxJdRul67Hkr5mDX8+F/1hrzP8EJy2+jrLVdLXElwcle7Mvs5yNdMXiyJ9Ta+3/a7916JcyWyhM6751+N5XJKX9q79V419eanpKF+uU33xpcjzj+38FxwAWu5oTrs90ddi7TZPqHURLyxxne3nFP2vRbkoCNPJ/HbB1UF/1QSjEpfgNO2vVnNJ/2vR/qoJb5W4Hvfp1Wz8WDfuEH3loeAc5xw3mc+1G07K73j8yFwV41p8ICvnWb3b8WMdlx3gejCdrP9VGwdgfS3MheMOybNq5b/q4yasr0XjJjYBk+/meYa1cabDmXjOOXEma2BKoZv8HI7LeUVcLpa4XJiG/Sbxwm7ymWrjmKSvrWZcbAQN/Vdt3HdOPJpLNcfqRl+BxO9tEb8XLsPx6O1mXO3sq3ZegToUT8vzClyq2WM312PtPAx1KLbL8zCiuJq/tBP/ZUcYN3HuIpJ5q6CYt6IG8kDm086bt+K/tBN/b8fINX+ejwKG8aLzfCydtI8m/8q9/QjmPr9OeF70tJgXxeu84bxoMltYTmLMPqiYRz50va+tJeeRTSf+i+bdA5l3t8W8e+y+j8CBPZ2Zdz+qaoZE6OnzbfVVm6cAF+T2TJ7CUb27N4bXvWtpX7V5HXBB5jN5HUeVbpXGtZxl2FZfXpEHE8/JgznsbVGOjFyFEXLN3xWvv5rSflvaV13ekJef9A+4brG8oXF399cWBwqlo+AXl1zR5oTS6arLs7LpzdWJvtrmf0V5V3lpxNXV/R3d5fExFw3W2tpXp3mPN0vrpgtO4/zVDvNESV/E9eg6vf7YlKvDvNou7atWvCdL/PL09djWvmp1sp3/t7Kugquz9QFqbOiSM/Kkoq6Kqyv/5RcOqejwRdLU1NXN49pY76x9NIFrh2Z9VGroZH3nBNMeoU76x67/U52HvAudX+5PtLWvKMXktLJPdwRhhhCHmPbo6oaYUweAGdfNkQHqtJv+F0YMMXoyaQMzDlRfgn4OBqqhgxZjnfsNW9WNjo+hRsaPLA39F+oKoyexNNcYG4Cv/dHm5uY2bBV9IFjKwVY5/OhZNtlvMltYTrhHb8p9LMNvGAh4SnUJdbRhJBBWGX5YQmhrXwFyTfVJMSEcrCQ8/GxtrQd1XwMX9leRa4FDte7fI9dUHx6vTnBDFMiEuhfAhf37Mf2Xuj8UQbxHN67jq6H/ipBrasyTwffw/svNzdubn96DYThyJeT2w9rxUEfrKcQYDRkbGUqnNPuEWqO4yZ9hTS80fLJE5ypqx4/8vKaW9sVRGiOhhwyjcwYWBbFv1q6atQ+34fkEMTkKn7h25u6K7wvoJJ5jmSuRENLABFSzYTyOyyWujFwQn0Cujap9AUMn/stjrlIsaZ1q1o3/9033eXkrdbpjBxYS1/oCXILTMN83p2yzVGJvQ7mXftUEbCCpszUwetcYofsal5ZzmBb8vpP4hHCVYoJ0V4s7nf5na+4oa73MZMQ1Eq6gam8lLsFpGF9lrlIMlY3aT0BfD93PwDLXmNzqWC6NM4IMPO7ok/u6/u2uuO7KMcLN2+7z8qd3bTrDVaUD+L6b5zWtR2j3ox12985jsHPy0ltOVzduOIfvcasdGzJ7cXHzuXiI186+rjHXzQlXRjU2/eZVLHy4c4bLVnDZCUNLfW0w14YvXPeFK9vtP97f3+/3v/KF675wZefuuKX/2mGua8Vc3oOUq7J7m/h5+aeBcD2o5+pwPfe7HP9an8wxyn4Grnl0gxrXQAbcavvPyex5QHBGpvK229mXcK2e5br785/Ah1372aJcHa7nPhCuULheFFwn/f39ZP9h/0+hcL2o5xqW593dpYzSzH9lzBUUXMdS9Yt/3cbPzR8XXMfCNX/kkfklrmS2sBwX56/6Z7luuu6EGy/f6D+9JsOOYzb7inzfrNQOtLSvGq4fvCH/tba1KFda0s3/AAAA///MnUFrHMkVgKu3hXoPkxmLEKKDPBP2F/iogFZjyBifTSJ08/oH7EGwOYhEaFp4yZqwoN1DrjHsKdiwvvpgkjby4svisLCGHIzpRYcFB5IOzkIflO10vVc1U9JUV9ebrmr1a7BG7tH0p6fXr16996q6YX/OjOtvkms22Xn/Tem+2Lv3Hjx6IrmkmzD1IUucB1/gsVy/XCK4whnX7J66+gy/rtx8LLmmBK744guU4qJUfJT86UUuvkznvXdK+3r4OBKGfyjM/scN/Yed05fevppzXX0p3rNrywV2X7O+w4m+7pWf+UdrfaGfkFwV/suBvp5dxxc3bbnQr5r7ya25Ku2e29cvGNiXnHYcCrNP9Vw4DgmupvZVfT++lP7LlgvHbSf990Z9/eVe+eVde31hnGPWV3MuxX9ZcqG40ZcYt/X29UXpv97j+hKGfyjMnllwNbSvai7Ff9lygW7c3I8Grrn/suUaK1zlXAqOJf2XgUv4L25fdlxBoXBJnCXtS8w79PrC+KvUlzD8Q2H2FVwD1U80ux9TwaWLc2bx1xPJVUgufaJpmsAXF+vTZlwjiaXEqzL+2pBc30uuTe0vKVTt4H40cf3yv9fh68quLVeqfNPsfmSnBeZN/r7Itf9GzB8fjcS0o/hemL2yr6PKpdYbGurrreB6MeOaz9N+uAVXW7s943p+X3DtaT8MKjU19VpLro8kl2Zey+eP9/j8cSC5TsxcUHmQfWnN9CW5XmvyAL/F/MTk9iJXRaKcl9xq9nu05DLlTX4n8l9PbPMmwCD7Hpvpy5Rnel/kvw6s80x8HJr1r15ncCynL1Neblvkvx7b5uXAtGr6fS25THnMIdjXymQxX1iRx4T70U2/b1+M23uavO9Q/MZZIKYd/dnEQ3st9F+O+qMFlzZPzvP3bG1nxjWs4UpVLvmWJesdd4HrqVJXEGPygEWYv38IHQCca4vX+oFL+1mor5r70VJC5DpR6kMihhmy6BlP4E9uJtwvca59XjviXPr6kKjMm/2XLVcC847yhwVXJi+6Ietp5S8sph175bnAUHiH+KvG31tKADW7rUhX5xP1x93yHHLxc8BV0YeM8aoYH5PrKL9aiotlwDXQ1UVFvfaRaJ/IeZkoDkwNFMr90LReuw9cQ20d+WAyWVmZ3IZemZIr5OeAq6qOzG3J0X5WePcdLNTdw/LfbfiFoSbPDf+YnxvNmmQqxI2/F7f8uT4F+CvxPoXRDu+fgHOc6z4/B1yJgUv6iY/ZChwXaoK2XNDlE+j7OqBg+zBDg46Kv/Jz1W5VSIh7RzXVV5Qy0Usm3Jfog+HdUtEPk8mNXTjHueAc5xprP0nKK+SSOMvFE3jPwzx5jG6iVBMnga532PeOn5v1DQ0M7kvU3XF8Jegr0vbVQNcNfzFCN4FrZHA9CuwTCOfUPquwwk2c56rwXxqusbYz0NSXNn7z4KF9X5rYV1H8He3911T7tzT18Q3+t/OBOGfTxwdDmLR7+aZ6/5VtHmr+110fMvYpkOOJIOlp+x6c9SEjl/Cr0ccrKFU9DXOuuB/p/n8g26bm5ZVpYXFOI+o4ZK2vMI689Cpf4Lr4svaaLXNZ+6+Wuaz9VwtcFvVaDVcy8M01ULjiiy+qJEj7tfdsIwnUjm6C/8q2q/q23Eigelx7/8WKs22PVKqPY6R4Yprr08hehBB/DdJrLXI1jFd9STlZR7nZFS6sLnROXyHGG03je+cSxZCoosy3Q2O/tSPpY0KI4L/GgzZ01jPXhzQyvV8dAbuTHrmeVrz2Ow6hkPUVfJdr42jHIriq/NeihEnmO87hQtZXGO+1wbUqnzs/u2zND7TERfZf3rlw/bbw9wT7aodLpAkI+koy73H03EES4nv/fmJTeY6ndTwRFK98+1WFixB/Fd7HoaX01cK4jVwJcMVXGBwW95r3OEflIsRf3gW5Uv6Pvf9qQZALEr+diu+RC2aDnYrvN/tKv699/qtNLnv/VbVIyjGXEIK+WpgNKVyfXUH5aS3X41a57PX1Z/9ccyHY13Gs/QQ/QtDX3bRNriMWwFHrv8KjqjK+K4F+8h4+do7iv6aLH+VUoP++j+MQwb7iiuVbzgSfdyLmaYT5UGizEUIDgfUdP4khn1Plv3RcWHL1J7AepheT59uV65vdiHjuQ2LMT+jsyycUk+uteneI/dFtcV1DrqMApd5/tcS1jnbfOX31odm8Q/l7Yfe4dWqX4nv0E6JP6/Mra3DU+i//cn49svX8cV3uXe1L1PXbhPnj/tjz+Giz3l1jX/nUc94E4pwgvgNc1v4ryHJ9n65bCWPifDtI0jby9xEj+q/wKPU8bsP+5KJuRfD3R4nnvC/s5y7rCp+vodTPH71zJeDvV6nxl3eubDDnIuTvfXOxnDeQ0vWV+Oba5h25vUjEX2sBHPX5e+9+AuZbqwPifCjI9jzn72H8ja5if7X9+Hi26bc/h0Up4x25/F9Sf47vGAz6YOX+mNb+i43M+4o3l+3l4onQ4rGzjUTt4+pSfJ9BvJLCNx2K78U+NWT78s4Vgw/9B3LZx/fMc3wf4P5fL+Cb6NvfoOzGNT8Wxr7je5TneDVCPsd3fI/yFEAI8VecV6x3cytJClyE/EQr8T1LqPnVo8RvfC+5qPlV73EhiKzzVdjXorTM1TV9Ydmd4r9a5aL4r3a4xNXs7Stvx0+Iq9nrq0g9x/fwFJfgD/A6+mpyA476+L7IPMf3sIFz+Ikxv6qRKPPcfz/la8WiVaL/Yuya5/77M75qsv+Og/1z3ErGVxH3QsxPWPsv7xKkfKGh4HIW30enR0WYjUdHxeg4P/1xzPbYafntcbHBxhuDZPSf50kdV8L7FCSXq/jeNRdFX2l7XNFXN1Bs+r/a4Fql5r9a4or6RvtaFL5Y1vAeB1xwP4Zn1Hyhby70X2ITiOileCpvffzlnQv8vbyafb4w92xfOD5KLvvx8cw3Fz4QAps0CPfj2DeXeJQeXIXgvwaxZy78nB61fzVK2+BaXcV5rf34GORtcC0xPh60yBWJhxjvXPBfOq6xby7o66Dry5gvdMHF9ytbIv4K2+QixBPGxw84sa/yAqsRrn+ssC+yOOHa43EO1N2dzYeccO3zOAf9aofie7xIfge4CPejsaPcCdc84U3wX9vGdTqOuSj1R+O6Jlf+Xu4L+83aLTh+XctVPDH157jmstZXzbo5x1z29hWY1xm64hpQ9RXGxnW/zrhSan+Oeb2os79j7nY9sjOuodG+Lo8r+hSuRtCXca2rA78aQ00h+Bqu9s0tlFr/VQZHfv1EGUbBQPchcNn7r7TyuWeOuDLc+tAYf2n8fc5M+XsHXOJZddR4db9iG3ZnXK+U/eejP/0M5ee1XOvMlL93wPVa2TC2Q/Fq8EJZN0eZP/rmes65xOSmS/n7k7jPy4lYt3p5aweODujrJOH5aOzjI+hr5NvfP037s75Hgn1NjXVkF3nybFjbv6rhKjzHX0GyvzHv963wX5pxKMt9c21tLaGv8sd8c/HGWqkva/sKk6FvLr6Qgt4fHRv3L3TBxRNZNfejjiu665VLfI7Zf+m4wpMWuEQfMsG+4uDULxcsRZZ9yIT5I3vrl2tLed4I5X5kH/nlOlCeG0PxX+z3frkgjg4+SeHj7PMTKe6r7Y8LnuMUHlPXP+bGDc+d1bc3cL2VfT5637hO2gXXesnV3yT2Y5bzDt/+fqM/W4/cofz9Oa4uxfc2+rpsrvCNkH9ePlc6LP1Ev3P6Yum49Kur68b78TK48ikvqnxq9F+XwTV9m/OqB+4T+OBLPDqgr/F3KZP76BLiicJ3f85AeQch/vLOde7jrP190CpXlf/SiHnVnAMuNSwgjI/ahyM65VLeQYgnzN3RLrhS5bW9vsyrh1xwKZYSfSnkUS1X33jWBdeB8tre35tXBbjgUuoDXRofI6VO3aXxMVIcRfQvIf92y/V/AAAA///snU9u4zYUxikQKLswrG2ACtYVulRRIzpGV4POEbIp4kVg0eh+TtAbFOgBJotR0P10VcymwfAEGW2KChjX7KP+xNTUcSiHjN6072NgGEbM/Pzl6fFJJsWTuKyJSaj8sjYwQxVfbD9/FdP5kP3hxS93bXs8f4mj67efaX7OAeX62Pra6ebnHNsBylN8Wc/dr+fURzdk883lnL+Cf799ol+8DHw9Z6BR11efZV5H192I69GhuWbWtu8Pxde/FZ5rme7HoTHfd4TmajaH7P+a+/cdweO++uqUfB8+T6iZNU/BOb6C59WonD0+f+KAQo9DUTm37of8utP1kOvA+Bh83La5RtSrweucARee+v5Uv56Vi//ca3IuphYo/WIqOSV/hedaLU/KX8G5itqKr+vXXZueK61w+mVfj8YUX4PuEPllC1P+4vb9ahHlr9QagBGNj4ONtDH5tbqw1klf95qeqzrbf0WAyS+VWPO28cTX51F/4YkvJ79GyzfX7q5tT91r4j/sl11HPxRfE3BBnth/lYjIL1Yvrbz64a5r03MV9X7eI6L8xfLKmo+JJ39BHf1y3x0ivwbd7TpNn7+G3SE6Hgf7gSHKXwzneqsh14deyLjw+BUph/iagmuL1C8tLa77Pzw5F0sVyvqL8Rpp/lrj9Iulj8fXJFzi1f4pJr+it/dPUcUXO2m+yTNw7SfMoYovhvN8aFh/fezaE7k8y5tfnuUtvjwothAw+dWuC2glrt90TU7G06tZR9EJk1/VpTW/EFF8qXPruq9Xv3LJZlDesbVJRcWWrSP4vHl/r9dHFKmFdb+Oj718cBVmaWVRQ0UMqbvYRnoDXEUpnDb+aNeBdfLrlza3wjVLVEoY6vRW6Bvg0irW47l8xlekKnYVVefiRgGXYuJHxTi8GDttsBHOL16u2DYq54JVEGJm/pNiX8CLC3Mjx5Fcb3r54JIZ33IZxzBo75i57XLFZvBicgKXV79kJv7gUpi9qu+a5cUXLIEXM+bGdW7VOT7jCxDin5p5qBfRW/DIpKOs4VIubw+WvwRL5knLxQ2XWcn4tTtXsHwPXF+2XIq/in4rs7UhLFeOXMHGR+Ay/7s540rMI119Ax9WQZ5w5BrUE579arlSGQNX/S3kV8W0cuQKVn91XFDRl/M5V1c5LyHKinJ59I6yh7sK4NeS5SqZc5lAzo/KSKvk6B14D3cVwK8VHFpmytRiCfEvuapT4cR1Zk3QCeFXBUdh1tyCAI5GaZLazolrldvzJzq988Zlgim76LgEE3Iptk5cdWHlCf9+8RK4qj0XS6LKiauq9gv6AsSXOdwzDSninuv4jhG9IqWsccjr+AgjT9JcZGi5zhj8Ow2XWz1xo6xx+/ZFq+99cMkMIJaQWIHrVwljZcuVOXKVgerVlmsF9eCKmfyVMGW4lqdw+a5XE0gTAuquuSnzIuAydaHThl3h/DL1valNxUYBl1rFvITDU9ULe+Rz5Pr9tm0+8hcMOcCltdm7YQ4nR0LLxNwgwfF8KJhfDA7ChGttzh/hvFZxbXKEVsJtE9BBnvB9vm242vPtVLKt4cql2/k2q14Gyl9P1NXKmj9xe/uiaT7y1xM1mPeIyK+43eqkEabrX9zyBpNftiC+Wr2XU6MMhNYvRPFlC61fFF+jRPE1ThRf4yT+vPyhaZdyapSB0PpF8TVK4t13neTUKAOh9Yvia5TEX5ed5NQoA6H1i+JrlCi+xkn8rduGjQurXxRfoyTe95JTowyE1i+Kr1EirnGC+OqanBplILR+PcyVs7jUVb6NS/jh2jyHxy3LefOiVlGdbrQq6nTH0k1tfqTQ8Lgzj6yozC/CO8yb2j7M+3TXh/nFTdPHTqi10LJ5hPeZR+gVK9fD+Yv8Ii4P8aW7howLq1/ENZKr6ISNC6tfxDWOq09g2Liw+kVclL+Ii7iI6//BRfmLuIiLuD5XLspfxEVcxHWc6+pTGuIiLuIiLuIiLuIiLuIiLuIiLuIiLuIiLuIiLuIirk/0DwAAAP//7J09b9tWFIbP9S16PZHtEKCDKhYdPXXUYEQe3B9QoEYnA/kJzGBEQ1DRU4v+DE+GA2QOkgBhkKFjJ4+Br6cCHRxmsoAyZM+hSEsxJPGjkigB70P4S4AuHtNHr97r5cILXvCCF7zgBS94wQte8IIXvOAFL3jBC17wghe84AUveMELXvCCF7zgBS94wQte8IIXvOAFL3htkRcAACwdq2KiR5SSlhOSdWp15KaxGnEOVjuAe1VeOs0+hS77RezlcozGOqF+1K4Xp7biT5bfAFTEX/sJe5mUhqM2vZwb1wTauqfRQ1e8iPY9OVTbBIN956Y9Ly/t6tBYh/we+4nXgD9+4Acjx6t0UuxqMHFHhZ7t0GCgAyNekQnoET9onYonxa4EFbHCQ/bq+ezlG3kNBGQ76m34pYrKn78q9Av2emqJeqQDRw4s5+9VKF5Gv2jPy7zukfVzr654hewVZF7mdYteHfY6yLwMdXznV/UuEkMtXp3Sp6+MnV32kr+dTx7PmJue/hWzoWtOQ7Oz256X3KjcK6YBe729StjLpCo0bVrdeVmVkO97+nrUJYd0oqy7CV7KqpRfAB265gxzyOUfvE3w0tmB5T7RR8vzT54JR/1N8OKQ16chez0OddCRg9WHt5vgxcOk3gW5V4/2le3/vQleXfb6c+LFD7q/bYLXU/FKkykvajknviEpzFHh5bOXn3k55c9dJTziHF6WfPHqkG/HXtfhJnhxTAz4g/PLck6wl2rdi6spl/yAety7uE9Y32Uv6YUtvmsLXOWJezTtc1T4rg4HXZ4tztWo5f8aubJPc9ORtHmfN0f9WOIsDXg/1CqGX4TWS0eyf+R9LXmyP+N9Wt+26yX7bfHK9ttcdkz2Nh7LfhsAANaGl9YlXLhe7eXSdOa7RH2vpbNVXsuoJjvC99Ps7e1dLOD58xsmSZPFXorUZ3w9i5+Eo7pcFudFv//0aZ33KxB+n+b8/HzRrbq4ePbslfBvY6+DMYf3+DGn8j07OTkpDi18crvO+WK+E6YG7OzsbNE9+0fm68OYuV5ffcas2XowpvZ0HR8fF8eRX12t7fW4S7vC1Gz9ISyerouXL7PxevOmkdcXBfen6/DnjBo37Rcmn67hcLjW+aobYHl+5QE230vdi7BZ8dUowC4vL1vJr4AaxNc4vyYBVtPrYG6AHdbLr6NJft2uO7/oXn6VBNh0fn2Y41U9vh7UnK5JfEl+zQ2wpd+v+/E1DrCy/Hr1P/KrCK8lxNfRJL6ezIwv9K8p0L/Qv9C/svxC/0L/qgr6V1PQv8pB/2oG+ldl0L+agf5VDvpXU9C/KoL+1RT0r3LQv5qB/lUZ9K9moH+Vg/7VFPSviqB/NQX9qxz0r2agf1VmZf3Lm/dbrA941WOrvEA9vLb/ils2X17bVnO8vk1UolIqrmGQX2E/vzxbXG6UXyOTXzrOL1lkfDVZCl7wWrdXV1a7Wyst1gqKtfp3a3nFWlGhZQqt+E6ryVIDeMELXvBq4rWpuQoveMELXtvqtal5Dy94LfD6DwAA///t2sEJADAMA7FRsv+Whe5QHBdpgnuZPKJL17V1V3Xp0qXL/aVLl65fu7buqi5dunS1dm3de126dOlyF+pKdk36u7Ds73HSVWVdAAAAAAAAAACPHVk+3tQ=:5361
^PQ1,0,1,Y^XZ';
END_VAR

//    Program: PRG_TCP_Client
//    Description: This provides TCP Comms to the zebra printer
//    
//    Created by: Ben Hess
//    Created Date: Tuesday, May 1, 2018

// Here's an example label

IF HMIData.printerSelection = LabelPrinterSelection.ZebraPrinter203DPI THEN 
	_sTCPSendData := label203;
ELSE
	_sTCPSendData := label300;
END_IF

_TCPClient_ipAddr.sAddr := _sClientIP; //set IP address
_TCPClient(
xEnable:= _sendLabel AND NOT _TCPWrite.xDone, // manually toggle for testing
xDone=> ,
xBusy=> ,
xError=> ,
ipAddr:= _TCPClient_ipAddr, 
uiPort:= _uiPort,
eError=> ,
hConnection=> _TCPConnection_hConnection);

// set TCP connection
_TCPConnection(
xEnable:= _TCPClient.xBusy AND NOT(_TCPConnection.xDone), //when server is ready
xDone=> , // client manually disconnected
xBusy=> ,
xError=> ,
hServer:=, // point all connections back to the same server
eError=> ,
xActive=> , 
hConnection=> );

// only execute on active connections

// write when connection is ready
_TCPWrite(
xExecute:= _sendLabel AND _TCPClient.xActive, //manually enable for testing
udiTimeOut:= 600000, //in microseconds => 600ms
xDone=> ,
xBusy=> , 
xError=> ,
hConnection := _TCPConnection_hConnection,
szSize := 25000, // write length only
pData := ADR(_sTCPSendData), 
eError=> );
//reset write enable
IF(_TCPWrite.xDone) THEN
	_TCPWriteEn:= FALSE;
	_sendLabel := FALSE;
END_IF

METHOD SendLabel
VAR_INPUT
END_VAR
_sendLabel := TRUE;
END_METHOD

END_FUNCTION_BLOCK

// FBs/Components/PrinterFB_Mode2
FUNCTION_BLOCK PrinterFB_Mode2 EXTENDS BaseComponentFB IMPLEMENTS IComponentStatus
VAR_INPUT
    autoSendLabel :BOOL;    // Automatically send a label
	ribbonEncoderPulse : BOOL;	// Ribbon Encoder Input
	enableRibbonDetection : BOOL := TRUE;                
END_VAR
VAR_OUTPUT
    state : PRINTER_STATES;         // Printer State Machine
	oLowerPrintHead : BOOL;
	printHeadDebounced : BOOL;
	ribbonFault : FB_Fault(name := 'Printer Ribbon Fault');
END_VAR
VAR
    _amPrintNow : BOOL;                // Auto mode - print now
    _amSendPrintSignal : BOOL;        // Auto mode - send print signal
    _amGoToIdle : BOOL;                // Auto mode - Acked, go back to idle mode
    printHeadDebounce : TON;
	printStarted : BOOL;
    printHeadDebouneSetpoint : TIME := T#50MS;
    tcpServer : FB_TCPClient();
	endOfPrintONS : Standard.F_TRIG();
	printerRibbonMovingTimer1 : Standard.TON;
	printerRibbonMovingTimer2 : Standard.TON;
	printerRibbonMovingSettleTime : TIME := T#450MS;
END_VAR

VAR_IN_OUT
END_VAR

//    Function Block: Printer
//    Description: This program manages the aspects of a (Zebra) printer
//    Created by: Ben Hess
//    Created Date: April 2nd, 2018
SUPER^();
// Enable TCP Server for label sending
tcpServer();
endOfPrintONS(CLK := printerEndOfPrint);
//Report as ready if mode is auto and we're not faulted
_ready := (_mode = DEVICE_MODES.Auto) AND NOT (state = PRINTER_STATES.Fault);

printerRibbonMovingTimer1(PT := printerRibbonMovingSettleTime);
printerRibbonMovingTimer2(PT := printerRibbonMovingSettleTime);

printHeadDebounce(PT:= printHeadDebouneSetpoint, Q=> printHeadDebounced);
printStarted := printerEndOfPrint;

IF enableONS.Q OR resetONS.Q THEN
    state := PRINTER_STATES.Idle;
	_reset := FALSE;
	_amGoToIdle := FALSE;
	_amSendPrintSignal := FALSE;
	_amPrintNow := FALSE;
	printHeadDebounced := FALSE;
	oRunPrinterRibbonUnwindMotor := FALSE;
	oLowerPrintHead := FALSE;
	printerRibbonMovingTimer1.IN := FALSE;
	printerRibbonMovingTimer2.IN := FALSE;
END_IF

IF NOT enable THEN
    state := PRINTER_STATES.Fault;
	oRunPrinterRibbonUnwindMotor := FALSE;
	oLowerPrintHead := FALSE;
END_IF

IF HMIData.printHeadServiceRaise THEN
	oLowerPrintHead := FALSE;
	HMIData.printHeadServiceRaise := FALSE;
ELSIF HMIData.printHeadServiceLower THEN
	oLowerPrintHead := TRUE;
	HMIData.printHeadServiceLower := FALSE;
END_IF


//State machine for the printer
CASE state OF
    PRINTER_STATES.Idle :                            //Go to waiting for data if printer is ready
                                                    oRunPrinterRibbonUnwindMotor := FALSE;
													oPrinterStartPrint := FALSE;
													printHeadDebounce.IN := FALSE;
													printHeadDebounced := FALSE;
													printerRibbonMovingTimer1.IN := FALSE;
													printerRibbonMovingTimer2.IN := FALSE;
													IF NOT printerDataReady THEN
                                                        IF autoSendLabel THEN
                                                            tcpServer.SendLabel();
                                                        END_IF
                                                        state := PRINTER_STATES.WaitingForData;
                                                    ELSE
                                                        state := PRINTER_STATES.DataReady;
                                                    END_IF
                                                    
                                        
    
    PRINTER_STATES.WaitingForData :                    //If printerDataReady drops out the label data was received
                                                    
                                                    IF printerDataReady THEN
                                                        state := PRINTER_STATES.DataReady;    
                                                    END_IF
                                                
    PRINTER_STATES.DataReady :                        // Wait for command to begin printing
                                                    IF NOT printerDataReady THEN
														state := PRINTER_STATES.Idle;
													END_IF
													IF _mode = DEVICE_MODES.Auto AND _amPrintNow THEN
                                                        state := PRINTER_STATES.BeginPrintCycle;
                                                        _amPrintNow := FALSE;
														printHeadDebounce.IN := TRUE;
                                                        oLowerPrintHead := TRUE;
                                                        oRunPrinterRibbonUnwindMotor := TRUE;
														//oPrinterStartPrint := TRUE;
                                                    END_IF                                    
            
    
    PRINTER_STATES.BeginPrintCycle :                // Start printing
                                                    
                                                    
                                                    IF _amSendPrintSignal THEN
                                                        oPrinterStartPrint := TRUE;
														
                                                        state := PRINTER_STATES.Printing;
                                                        printHeadDebounce.IN := FALSE;
                                                        _amSendPrintSignal := FALSE;
                                                    END_IF                                                    
                                        
    
    PRINTER_STATES.FeedAtPrintSpeed :                //

                                                    
                                                                                                
                                        
    PRINTER_STATES.Printing :                        //While printing, wait for End of Print signal
													printerRibbonMovingTimer1.IN := ribbonEncoderPulse;
													printerRibbonMovingTimer2.IN := NOT ribbonEncoderPulse;
                                                    IF endOfPrintONS.Q OR printerRibbonMovingTimer1.Q OR printerRibbonMovingTimer2.Q THEN
                                                        oPrinterStartPrint := FALSE;
                                                        oLowerPrintHead := FALSE;
														IF printerRibbonMovingTimer1.Q OR printerRibbonMovingTimer2.Q THEN
															ribbonFault.Trigger();
														END_IF
														printerRibbonMovingTimer1.IN := FALSE;
														printerRibbonMovingTimer2.IN := FALSE;
														 
                                                        //oRunPrinterRibbonUnwindMotor := FALSE;
                                                        state := PRINTER_STATES.DonePrinting;    
                                                    END_IF
                                        
    PRINTER_STATES.DonePrinting :                    //Done printing, feed a little more through
                                                    IF _mode = DEVICE_MODES.Auto AND _amGoToIdle THEN
                                                        oRunPrinterRibbonUnwindMotor := FALSE;
                                                        state := PRINTER_STATES.Idle;
                                                        _amGoToIdle := FALSE;
														HMIData.printerCycles.Increment();
														HMIData.printHeadClean.Increment();
                                                        Globals.printerCycleCounts := Globals.printerCycleCounts + 1;
                                                    END_IF
        
    PRINTER_STATES.FeedThrough :                        
                                        
    PRINTER_STATES.Ready :                        
                                        
    PRINTER_STATES.Fault :                        
                                        
END_CASE

METHOD AutoSendPrintSignal
VAR_INPUT
END_VAR
_amSendPrintSignal := TRUE;
END_METHOD

METHOD AutoPrintNow
VAR_INPUT
END_VAR
_amPrintNow := TRUE;
END_METHOD

METHOD AutoAckPrintDone
VAR_INPUT
END_VAR
_amGoToIdle := TRUE;
END_METHOD

PROPERTY Ready : BOOL
SET
_ready := Ready;
END_SET
GET
Ready := _ready;
END_GET
END_PROPERTY

PROPERTY Mode : DEVICE_MODES
SET
_mode := Mode;
END_SET
GET
Mode := _mode;
END_GET
END_PROPERTY

END_FUNCTION_BLOCK

// FBs/Components/MonostableMultivibratorFB
FUNCTION_BLOCK MonostableMultivibratorFB EXTENDS BaseComponentFB
VAR_INPUT
END_VAR
VAR_OUTPUT
	Q : BOOL;   // Output pulse
END_VAR
VAR
	_trigger : BOOL;
	_dwellTimeInMS : UINT := 80; 	// Pulse Dwell in mS 
	_delayTimeInMS : UINT; 			// Delay before Pulse in mS
	_manualOn : BOOL;
	_manualOff : BOOL;
	active : BOOL;
	dwellTimer : Standard.TON;
	delayTimer : Standard.TON;
END_VAR


// HPA is on for only as long as its setpoint.

delayTimer(IN := _trigger AND NOT dwellTimer.Q, PT := UINT_TO_TIME(_delayTimeInMS));
dwellTimer(IN := delayTimer.Q AND NOT dwellTimer.Q, PT := UINT_TO_TIME(_dwellTimeInMS));

Q:= delayTimer.Q OR _manualOn;

IF dwellTimer.Q OR _reset THEN
	active := FALSE;
	_trigger := FALSE;
	_manualOn := FALSE;
	_manualOff := FALSE;
END_IF

SUPER^();

PROPERTY DelaySetting : UINT
GET
DelaySetting := _delayTimeInMS;
END_GET
SET
_delayTimeInMS := DelaySetting;
END_SET
END_PROPERTY

METHOD Trigger
VAR_INPUT
END_VAR
_trigger := TRUE;
END_METHOD

METHOD ManualOn
VAR_INPUT
END_VAR
_manualOn := TRUE;
_manualOff := FALSE;
END_METHOD

METHOD ManualOff : BOOL
VAR_INPUT
END_VAR
_manualOn := FALSE;
_manualOff := TRUE;
END_METHOD

PROPERTY DwellSetting : UINT
SET
_dwellTimeInMS := DwellSetting;
END_SET
GET
DwellSetting := _dwellTimeInMS;
END_GET
END_PROPERTY

END_FUNCTION_BLOCK

// FBs/Components/DelayDwellFB/DelayDwellFB
FUNCTION_BLOCK DelayDwellFB EXTENDS BaseComponentFB
VAR_INPUT
END_VAR
VAR_OUTPUT
	Q : BOOL;   // Output pulse
END_VAR
VAR
	_trigger : BOOL;
	_dwellTimeInMS : DINT := 80; 	// Pulse Dwell in mS 
	_delayTimeInMS : DINT; 			// Delay before Pulse in mS
	_manualOn : BOOL;
	_manualOff : BOOL;
	active : BOOL;
	dwellTimer : Standard.TON;
	delayTimer : Standard.TON;
	state : DELAY_DWELL_STATES;
END_VAR

//    Function Block: DelayDwellFB
//    Description: On Trigger(), starts a delay then sets the Q output for a dwell time.  Each addition Trigger() resets the dwell timer.
//    Created by: Ben Hess
//    Created Date: February 20th, 2020

// Setup timers for reading offset and scanning distance
delayTimer(PT := UDINT_TO_TIME(_delayTimeInMS));
// If negative dwell time, run forever
IF _dwellTimeInMS < 0 THEN
	dwellTimer(PT := T#0MS);
ELSE
	dwellTimer(PT := UDINT_TO_TIME(_dwellTimeInMS));
END_IF

// Manual On/Off
IF _manualOff THEN
	THIS^.Reset();
	state := DELAY_DWELL_STATES.Idle;
ELSIF _manualOn THEN
	THIS^.Reset();
	Q := TRUE;
	state := DELAY_DWELL_STATES.Idle;
END_IF

CASE state OF
	DELAY_DWELL_STATES.Idle:  			//
										dwellTimer.IN := FALSE;
										delayTimer.IN := FALSE;
										
										IF _trigger THEN
											IF _delayTimeInMS <> 0 THEN
												state := DELAY_DWELL_STATES.Delay;
											ELSE
												state := DELAY_DWELL_STATES.Dwell;
											END_IF
											_trigger := FALSE;
										END_IF
	
	DELAY_DWELL_STATES.Delay: 			//
										delayTimer.IN := TRUE;
										IF delayTimer.Q THEN
											delayTimer.IN := FALSE;
											state := DELAY_DWELL_STATES.Dwell;
										END_IF
	
	DELAY_DWELL_STATES.Dwell: 			//
										Q := TRUE;
										IF _dwellTimeInMS >= 0 THEN
											dwellTimer.IN := TRUE;
											IF dwellTimer.Q THEN
												dwellTimer.IN := FALSE;
												Q := FALSE;
												state := DELAY_DWELL_STATES.Idle;
											END_IF
										END_IF
										IF _trigger THEN
											_trigger := FALSE;
											state := DELAY_DWELL_STATES.ResettingDwell;
										END_IF
										
	DELAY_DWELL_STATES.ResettingDwell: 	//
										dwellTimer.IN := FALSE;
										state := DELAY_DWELL_STATES.Dwell;
END_CASE

SUPER^();

METHOD Reset : BOOL
VAR_INPUT
END_VAR
active := FALSE;
_trigger := FALSE;
_manualOn := FALSE;
_manualOff := FALSE;
Q := FALSE;
state := DELAY_DWELL_STATES.Idle;
END_METHOD

METHOD ManualOff : BOOL
VAR_INPUT
END_VAR
_manualOn := FALSE;
_manualOff := TRUE;
END_METHOD

METHOD ManualOn
VAR_INPUT
END_VAR
_manualOn := TRUE;
_manualOff := FALSE;
END_METHOD

METHOD Trigger
VAR_INPUT
END_VAR
_trigger := TRUE;
END_METHOD

PROPERTY DwellSetting : DINT
GET
DwellSetting := _dwellTimeInMS;
END_GET
SET
_dwellTimeInMS := DwellSetting;
END_SET
END_PROPERTY

PROPERTY DelaySetting : DINT
SET
_delayTimeInMS := DelaySetting;
END_SET
GET
DelaySetting := _delayTimeInMS;
END_GET
END_PROPERTY

END_FUNCTION_BLOCK

// FBs/Components/BagOpenFingersWithSensorsFB
FUNCTION_BLOCK BagOpenFingersWithSensorsFB EXTENDS BagOpenFingersFB
VAR_INPUT
	rightFingerBagPresent : BOOL;
	leftFingerBagPreset : BOOL;
END_VAR
VAR_IN_OUT
	bagFailedToGrabBothFingersCount : UDINT; // Both Fingers failed to grab bag
	bagFailedToGrabRightFingerCount : UDINT; // Right Bag Open Finger Failed to Grab Bag
	bagFailedToGrabLeftFingerCount : UDINT; // Left Bag Open Finger Failed to Grab Bag
	successfulBagOpenCount : UDINT;			// Successful Bag Open Count
END_VAR
VAR_OUTPUT
	
END_VAR

SUPER^();

METHOD CheckIfBagGrabbed : BOOL
VAR_INPUT
	incrementCounters : BOOL; // IF TRUE Incerment bag counters, otherwise just return bag grabbed status
END_VAR
// Returns true if bag grab successful.  Also increments appropriate counters

{warning disable C0371}
// Checking the VAR_IN_OUT reference, leave the current method in case of invalid reference
IF NOT __ISVALIDREF(successfulBagOpenCount) 
	OR NOT __ISVALIDREF(bagFailedToGrabLeftFingerCount)
	OR NOT __ISVALIDREF(bagFailedToGrabRightFingerCount)
	OR NOT __ISVALIDREF(bagFailedToGrabBothFingersCount)
	THEN RETURN;    
END_IF

IF rightFingerBagPresent AND leftFingerBagPreset THEN
	IF incrementCounters THEN
		successfulBagOpenCount := successfulBagOpenCount +1;
	END_IF
	CheckIfBagGrabbed := TRUE;
ELSIF rightFingerBagPresent AND NOT leftFingerBagPreset THEN
	IF incrementCounters THEN
		bagFailedToGrabLeftFingerCount := bagFailedToGrabLeftFingerCount +1 ;
	END_IF
ELSIF NOT rightFingerBagPresent AND leftFingerBagPreset THEN
	IF incrementCounters THEN
		bagFailedToGrabRightFingerCount := bagFailedToGrabRightFingerCount + 1;
	END_IF
ELSE
	IF incrementCounters THEN
		bagFailedToGrabBothFingersCount := bagFailedToGrabBothFingersCount + 1;
	END_IF
END_IF
{warning restore C0371}
END_METHOD

END_FUNCTION_BLOCK

// FBs/Components/BagOpenFingersFB
FUNCTION_BLOCK BagOpenFingersFB EXTENDS BaseComponentFB
VAR_INPUT

END_VAR
VAR_IN_OUT

END_VAR
VAR_OUTPUT
    releaseOutput : BOOL;
	grabOutput : BOOL;
END_VAR
VAR
    _releaseCommand : BOOL;
    _grabCommand : BOOL;
END_VAR

SUPER^();
releaseOutput := _releaseCommand AND enable;
grabOutput := _grabCommand AND enable;

METHOD Release
VAR_INPUT
END_VAR
_releaseCommand := TRUE;
_grabCommand := FALSE;
END_METHOD

METHOD Grab
VAR_INPUT
END_VAR
_releaseCommand := FALSE;
_grabCommand := TRUE;
HMIData.bagOpenFingerCycles.Increment();
END_METHOD

END_FUNCTION_BLOCK

// FBs/Motors/Applied Motion/FB_AppliedMotionStepServoEIPPassthrough
FUNCTION_BLOCK FB_AppliedMotionStepServoEIPPassthrough EXTENDS FB_AppliedMotionStepServoEIPBase
VAR_INPUT
END_VAR
VAR_OUTPUT
END_VAR
VAR
	homingState : JAW_HOMING_STATES;
	homeRequiredONS : R_TRIG;
	timerHomeDelay : TON;
END_VAR

SUPER^();

METHOD HomeNow
_homeNow := TRUE;
END_METHOD

METHOD DoneClamping
VAR_INPUT
END_VAR
sclCommand := 16#434D; // CM Control Mode
parameter1 := 21;
															
commandSuccessful := FALSE;
commands.SendHostCommand := TRUE;
END_METHOD

METHOD AllowClamping
VAR_INPUT
END_VAR
sclCommand := 16#434D; // CM Control Mode
parameter1 := 1;
															
commandSuccessful := FALSE;
commands.SendHostCommand := TRUE;
END_METHOD

//{warning 'add method implementation '}
METHOD Stop
commandSuccessful := FALSE;
commands.StopCrash := TRUE;
END_METHOD

METHOD SetPositionLimit
VAR_INPUT
	positionLimit : DINT;
END_VAR
sclCommand := 16#5046; // PF (Position Fault)
parameter1 := positionLimit;
															
commandSuccessful := FALSE;
commands.SendHostCommand := TRUE;
END_METHOD

METHOD Execute
VAR_INPUT
END_VAR
SUPER^.Execute();
timerHomeDelay();
homeRequiredONS(CLK := homeRequiredIndication);

//IF _reset OR homeRequiredONS.Q THEN
IF _reset THEN
	homingState := JAW_HOMING_STATES.Idle;
	_homeNow := FALSE;
	timerHomeDelay.IN := FALSE;
END_IF

CASE homingState OF
	JAW_HOMING_STATES.Idle:						IF _homeNow THEN
													//IF NOT driveInputs[10].2 THEN
													//	homingState := JAW_HOMING_STATES.MoveForwardFromSensor;
													//ELSE 
														homingState := JAW_HOMING_STATES.StartHoming;
													//END_IF
													_homeNow := FALSE;
												END_IF
												
	JAW_HOMING_STATES.MoveForwardFromSensor:	commandSuccessful := FALSE;
												velocitySetpoint := 2583;
												pointToPointAccelSetpoint := 1000;
												pointToPointDecelSetpoint := 1000;
												distanceToMoveInSteps := -4000;
												commands.FeedToLength := TRUE;
												homingState := JAW_HOMING_STATES.MovingForwardFromSensor;
												
	JAW_HOMING_STATES.MovingForwardFromSensor:	timerHomeDelay.PT := T#200MS;
												timerHomeDelay.IN := TRUE;
												IF timerHomeDelay.Q THEN
													IF (NOT Moving AND InPosition) THEN
														homingState := JAW_HOMING_STATES.StartHoming;
														timerHomeDelay.IN := FALSE;
                                                       END_IF
												END_IF
												
	JAW_HOMING_STATES.StartHoming:				commandSuccessful := FALSE;
												velocitySetpoint := 1250;
												pointToPointAccelSetpoint := 10;
												pointToPointDecelSetpoint := 10;
												distanceToMoveInSteps := 1;
												ExecuteStoredProgram(2);
												homingState := JAW_HOMING_STATES.Homing;
												
	JAW_HOMING_STATES.Homing:					timerHomeDelay.PT := T#200MS;
												timerHomeDelay.IN := TRUE;
												IF timerHomeDelay.Q THEN
													IF (NOT SUPER^.Homing) THEN
														homingState := JAW_HOMING_STATES.HomeComplete;
														timerHomeDelay.IN := FALSE;
                                                       END_IF
												END_IF 
												
	JAW_HOMING_STATES.HomeComplete:				//MoveToPosition(2, 1000,1000,2583);
												homingState := JAW_HOMING_STATES.SetLimits;

	JAW_HOMING_STATES.MovingToTwoInches : 		timerHomeDelay.PT := T#200MS;
												timerHomeDelay.IN := TRUE;
												IF timerHomeDelay.Q THEN
													IF (NOT Moving AND InPosition) THEN
														homingState := JAW_HOMING_STATES.SetLimits;
														timerHomeDelay.IN := FALSE;
                                                       END_IF
												END_IF 
												
	JAW_HOMING_STATES.SetLimits :				commandSuccessful := FALSE;
												ExecuteStoredProgram(3);
												homingState := JAW_HOMING_STATES.Idle;
												
	
END_CASE
END_METHOD

END_FUNCTION_BLOCK

// FBs/Components/AdjustablePassthroughFB
FUNCTION_BLOCK AdjustablePassthroughFB EXTENDS BaseComponentFB IMPLEMENTS IComponentStatus
VAR_INPUT
	pressureBarEndStopMotor : IPositionableMotor;
	jogInPB : BOOL;
	jogOutPB : BOOL;
END_VAR
VAR_OUTPUT
    homeRequired : BOOL; //Homing Required
    passthroughPosition : REAL;
    state : PASSTHROUGH_SERVO_STATES := PASSTHROUGH_SERVO_STATES.Idle; //State indication of Jaw Passthrough Servo
    exhaustPressureBarRequest : BOOL; // Exhaust pressure bar request for passthrough movement
    extendPressureBarRequest : BOOL; // Extend pressure bar request for passthrough movement
END_VAR
VAR        
    passthroughSetpoint : REAL;        // Passthrough setpoint in inches
	passthroughTravel : REAL;				// Passthrough travel total
	capturePassthroughPos : REAL;
    mustMovePassthroughOut : BOOL; //Flag to tell us that the setpoint requires us to move the passthrough out
    _homeEndStop : BOOL;            // Home End Stop Command
    _movePassthrough  : BOOL;        // Move Passthrough
    _ackRequest : BOOL;                // Request Acknowledged from controller
	passthroughSettingLast : REAL;
	timerHomeDelay : TON;
	faultONS : FB_ONS;
	jogInONS : FB_ONS;
	jogOutONS : FB_ONS;
	
END_VAR
VAR_IN_OUT
	cumulativeChangeCount : DINT;
	cumulativeChangeDistance : UDINT;
END_VAR

//    Function Block: AdjustablePassthroughFB
//    Description:      The adjustable passthrough on the pneumatic head uses a closed loop stepper motor to 
//                    move the end stop for the jaw cylinders
//    Created by: Ben Hess
//    Created Date: Thursday, May 10, 2018
SUPER^();
jogInONS(CLK := jogInPB);
jogOutONS(CLK := jogOutPB);
//Add 2 inch offset
passthroughPosition :=  (pressureBarEndStopMotor.CurrentPosition) - HMIData.passthroughOffset;
timerHomeDelay();
faultONS(CLK := HMIData.faultActive);


//Go to idle when enabled
enableONS(CLK := enable);
IF enableONS.Q OR resetONS.Q THEN    
    state := PASSTHROUGH_SERVO_STATES.Idle;
	_movePassthrough := FALSE;
	Globals.jawMovingIn := FALSE;
	 _homeEndStop := FALSE;
	 timerHomeDelay.IN := FALSE;
	passthroughSetpoint := HMIData.passthroughSetting + HMIData.passthroughOffset ;
END_IF

IF NOT enable THEN
    state := PASSTHROUGH_SERVO_STATES.Idle;
	_movePassthrough := FALSE;
	_homeEndStop := FALSE;
END_IF

_ready := (_mode = DEVICE_MODES.Auto) AND NOT (state = PASSTHROUGH_SERVO_STATES.Fault);
IF faultONS.OSR THEN
	pressureBarEndStopMotor.Stop();
	state := PASSTHROUGH_SERVO_STATES.Idle;
END_IF

CASE state OF
    PASSTHROUGH_SERVO_STATES.Idle :                     // Go to ready state if no home required.  Otherwise go to ready if enabled. Stay in Idle if disabled.
                                                        extendPressureBarRequest := FALSE;
                                                        exhaustPressureBarRequest := FALSE;
														timerHomeDelay.IN := FALSE;
                                                        IF enable AND pressureBarEndStopMotor.HomeRequired THEN
                                                            state := PASSTHROUGH_SERVO_STATES.HomingRequired;
                                                        ELSIF enable THEN
                                                            state := PASSTHROUGH_SERVO_STATES.Ready;
                                                        END_IF
                                                        
    PASSTHROUGH_SERVO_STATES.HomingRequired :            //When Home Servo Pushbitton is pressed
														homeRequired := TRUE;
                                                        IF _homeEndStop THEN
                                                            state := PASSTHROUGH_SERVO_STATES.StartHoming;
                                                        END_IF
                                                        
    PASSTHROUGH_SERVO_STATES.StartHoming :                
                                                        // Start motor homing sequence
                                                        exhaustPressureBarRequest := TRUE;
														Globals.jawMovingIn := TRUE;
														//extendPressureBarRequest := TRUE;
                                                        IF _ackRequest THEN
															pressureBarEndStopMotor.HomeNow();
                                                            exhaustPressureBarRequest := FALSE;
															//extendPressureBarRequest := FALSE;
                                                            _ackRequest := FALSE;
                                                            state := PASSTHROUGH_SERVO_STATES.Homing;    
                                                        END_IF        

    
    PASSTHROUGH_SERVO_STATES.Homing :                    //Move on to Home Complete once finished
														
														timerHomeDelay.PT := T#200MS;
														timerHomeDelay.IN := TRUE;
														IF NOT iPassthroughHomeSensorClear THEN
															extendPressureBarRequest := TRUE;
															Globals.jawMovingIn := FALSE;
														END_IF
														
														IF _ackRequest THEN 
															extendPressureBarRequest := FALSE;
														END_IF 
														
														IF timerHomeDelay.Q THEN
															IF (NOT pressureBarEndStopMotor.HomeRequired) THEN
																state := PASSTHROUGH_SERVO_STATES.HomeComplete;
																extendPressureBarRequest := FALSE;
																_ackRequest := FALSE;
																timerHomeDelay.IN := FALSE;
                                                        	END_IF
														END_IF
                                                        
    
    PASSTHROUGH_SERVO_STATES.HomeComplete :             //Move on to Ready State once supervisor acks the cylinder request
                                                        _homeEndStop := FALSE;
														Globals.jawMovingIn := FALSE;
                                                        extendPressureBarRequest := TRUE;
														homeRequired := FALSE;
                                                        IF _ackRequest THEN
                                                            extendPressureBarRequest := FALSE;
                                                            _ackRequest := FALSE;
                                                            state := PASSTHROUGH_SERVO_STATES.Ready;    
                                                        END_IF
                                                        
    PASSTHROUGH_SERVO_STATES.MovePassthroughOut :        // Move passthrough out
                                                        extendPressureBarRequest := TRUE;
                                                        IF _ackRequest THEN
                                                            pressureBarEndStopMotor.MoveToPosition(position := (passthroughSetpoint + HMIData.passthroughOffset), 
                                                                                    acceleration := 150, 
                                                                                    deceleration := 150, 
                                                                                    velocity := 2583);
                                                            //
                                                            extendPressureBarRequest := FALSE;
                                                            _ackRequest := FALSE;
                                                            state := PASSTHROUGH_SERVO_STATES.MovingPassthroughOut;        
                                                        END_IF
                                                        

                                                    
                                                        
    PASSTHROUGH_SERVO_STATES.MovingPassthroughOut :        //Move on to Passthrough Moved Out once position reached
														timerHomeDelay.PT := T#200MS;
														timerHomeDelay.IN := TRUE;
														IF timerHomeDelay.Q THEN
															IF (REAL_TO_INT((passthroughSetpoint + HMIData.passthroughOffset)*100) = REAL_TO_INT(passthroughPosition*100)) THEN
																state := PASSTHROUGH_SERVO_STATES.PassthroughMovedOut;
																timerHomeDelay.IN := FALSE;
															END_IF
															
															IF jogOutONS.OSF THEN
																passthroughTravel := ABS(capturePassthroughPos - passthroughPosition);
																pressureBarEndStopMotor.Stop();
																Globals.passthroughChangedFromJog := TRUE;
																state := PASSTHROUGH_SERVO_STATES.PassthroughMovedOut;
															END_IF
														END_IF
    PASSTHROUGH_SERVO_STATES.PassthroughMovedOut :       
														extendPressureBarRequest := TRUE; 
                                                         IF _ackRequest THEN
                                                            extendPressureBarRequest := FALSE;
                                                            _movePassthrough := FALSE;
                                                            _ackRequest := FALSE;
															HMIData.passthroughChanges.Increment();
                                                            cumulativeChangeCount := cumulativeChangeCount + 1;
															cumulativeChangeDistance := cumulativeChangeDistance + REAL_TO_UDINT((passthroughTravel * 10));
                                                            state := PASSTHROUGH_SERVO_STATES.Ready;    
                                                        END_IF
                                                        
    PASSTHROUGH_SERVO_STATES.MovePassthroughIn :        
                                                        exhaustPressureBarRequest := TRUE;
														Globals.jawMovingIn := TRUE;
                                                        IF _ackRequest THEN
                                                            pressureBarEndStopMotor.MoveToPosition(position := (passthroughSetpoint + HMIData.passthroughOffset), 
                                                                                    acceleration := 150, 
                                                                                    deceleration := 150, 
                                                                                    velocity := 2583);
                                                            //
                                                            exhaustPressureBarRequest := FALSE;
                                                            _ackRequest := FALSE;
                                                            state := PASSTHROUGH_SERVO_STATES.MovingPassthroughIn;        
                                                        END_IF
                                                    
                                                        
    PASSTHROUGH_SERVO_STATES.MovingPassthroughIn :        //Move on to Passthrough Moved In once position reached
														timerHomeDelay.PT := T#200MS;
														timerHomeDelay.IN := TRUE;
														IF timerHomeDelay.Q THEN
															IF (REAL_TO_INT((passthroughSetpoint + HMIData.passthroughOffset)*100) = REAL_TO_INT(passthroughPosition*100)) THEN
																state := PASSTHROUGH_SERVO_STATES.PassthroughMovedIn;
																timerHomeDelay.IN := FALSE;
															END_IF
															
															IF jogInONS.OSF THEN
																passthroughTravel := ABS(capturePassthroughPos - passthroughPosition);
																pressureBarEndStopMotor.Stop();
																Globals.passthroughChangedFromJog := TRUE;
																state := PASSTHROUGH_SERVO_STATES.PassthroughMovedIn;
															END_IF
                                                        END_IF
    PASSTHROUGH_SERVO_STATES.PassthroughMovedIn :        
                                                        extendPressureBarRequest := TRUE;
														Globals.jawMovingIn := FALSE;
                                                        IF _ackRequest THEN
                                                            extendPressureBarRequest := FALSE;
                                                            _movePassthrough := FALSE;
                                                            _ackRequest := FALSE;
															HMIData.passthroughChanges.Increment();
                                                            cumulativeChangeCount := cumulativeChangeCount + 1;
															cumulativeChangeDistance := cumulativeChangeDistance + REAL_TO_UDINT((passthroughTravel * 10));
                                                            state := PASSTHROUGH_SERVO_STATES.Ready;    
                                                        END_IF
                                                        
                                                        
